// take a position and return always a positive integer between 0 and MAX_TRACK_LENGTH
METHOD PRIVATE TO_POS : DINT
VAR_INPUT
	pos : LREAL;
END_VAR
IF pos < 0 THEN
    TO_POS := LREAL_TO_DINT(pos + CONST.MAX_TRACK_LENGTH);

ELSIF pos >= CONST.MAX_TRACK_LENGTH THEN
    TO_POS := LREAL_TO_DINT(pos) MOD LREAL_TO_DINT(CONST.MAX_TRACK_LENGTH);

ELSE
    TO_POS := LREAL_TO_DINT(pos);

END_IF
END_METHOD

METHOD ToString : STRING
VAR_INPUT
END_VAR
ToString := CONCAT('FB_Mover_', TO_STRING(THIS^._iID));
END_METHOD

END_FUNCTION_BLOCK

// ---- POUs/20_AUTO/Mover/FB_Station.TcPOU
{attribute 'reflection'}
FUNCTION_BLOCK FB_Station IMPLEMENTS IStation, IObject
VAR_INPUT
END_VAR
VAR_OUTPUT
END_VAR
VAR
    _Position          : REFERENCE TO FB_Position;
    _Process           : REFERENCE TO FB_AUT_ABSTRACT;
    _WaitPosOffset     : LREAL; // offset of the station position, should always be negative
    _iMaxWaitingMovers : INT;   // Maximum of waiting mover in front of the station
    _iGroupNumber      : INT;   // The current group member
    _lrOffset          : LREAL; // offset position of this station for a given recipe
    _bSuperTrackNumber : BYTE;  // target number in superTrack

    _ApproachScenario : ApproachScenario_e := ApproachScenario_e.WaitOnFinishedProcess;

    _iID : INT := 0; // instance ID, is set during FB_Init using the value of _iInstanceCounter 
END_VAR
VAR_STAT
    _iInstanceCounter : INT := 1; // instance counter
END_VAR

PROPERTY ApproachScenario : ApproachScenario_e
GET
ApproachScenario := THIS^._ApproachScenario;
END_GET
SET
THIS^._ApproachScenario := ApproachScenario;
END_SET
END_PROPERTY

METHOD Equals : BOOL
VAR_INPUT
    object : ANY;
END_VAR
Equals := THIS = object.pValue;
END_METHOD

METHOD FB_init : BOOL
VAR_INPUT
    bInitRetains      : BOOL; // if TRUE, the retain variables are initialized (warm start / cold start)
    bInCopyCode       : BOOL; // if TRUE, the instance afterwards gets moved into the copy code (online change)
    Position          : REFERENCE TO FB_Position;
    Process           : REFERENCE TO FB_AUT_ABSTRACT;
    WaitPosOffset     : LREAL;
    ApproachScenario  : ApproachScenario_e;
    iMaxWaitingMovers : INT;
	bSuperTrackNumber : BYTE;
END_VAR
THIS^._iID               := THIS^._iInstanceCounter;
THIS^._iInstanceCounter  := THIS^._iInstanceCounter + 1;
THIS^._Position          REF= Position;
THIS^._Process           REF= Process;
THIS^._WaitPosOffset     := WaitPosOffset;
THIS^._ApproachScenario  := ApproachScenario;
THIS^._iMaxWaitingMovers := iMaxWaitingMovers;
THIS^._bSuperTrackNumber := bSuperTrackNumber;
END_METHOD

// the maxuimum number of waiting movers at the front of the station
PROPERTY iMaxWaitingMovers : INT
GET
iMaxWaitingMovers := THIS^._iMaxWaitingMovers;
END_GET
SET
THIS^._iMaxWaitingMovers := iMaxWaitingMovers;
END_SET
END_PROPERTY

PROPERTY PUBLIC Offset : LREAL
GET
Offset := THIS^._lrOffset;
END_GET
SET
THIS^._lrOffset := Offset;
END_SET
END_PROPERTY

PROPERTY Position : REFERENCE TO FB_Position
GET
Position REF=_Position;
END_GET
SET
_Position REF=Position;
END_SET
END_PROPERTY

PROPERTY Process : REFERENCE TO FB_AUT_ABSTRACT
GET
Process REF=_Process;
END_GET
SET
_Process REF= Process;
END_SET
END_PROPERTY

METHOD SetWaitPosOffset : REFERENCE TO FB_Station
VAR_INPUT
	WaitPosOffset : LREAL; // offset position from the given station, must be negative
END_VAR
IF _WaitPosOffset < 0 THEN
    _WaitPosOffset := WaitPos;
END_IF

SetWaitPosOffset REF= THIS^;
END_METHOD

PROPERTY SuperTrackNumber : BYTE
GET
SuperTrackNumber := THIS^._bSuperTrackNumber;
END_GET
END_PROPERTY

METHOD ToString : STRING
VAR_INPUT
END_VAR
VAR_INST
END_VAR
ToString := CONCAT('FB_Station_', TO_STRING(THIS^._iID));
END_METHOD

PROPERTY PUBLIC WaitPos : LREAL
GET
WaitPos := _WaitPosOffset + this^._Position.lrWorkPosition;
END_GET
SET
IF WaitPos < THIS^._Position.lrWorkPosition THEN
    _WaitPosOffset := WaitPos - THIS^._Position.lrWorkPosition;
END_IF
END_SET
END_PROPERTY

END_FUNCTION_BLOCK

// ---- POUs/20_AUTO/Mover/FB_Position.TcPOU
(*
    1D Position class, used to express a given position
	Since the position is in lreal format, you should
	always give a left and a right margin so the isInPosition
	flag will stay stable (beacause we cannot use the = 
	operator on lreal! )
*)
FUNCTION_BLOCK FB_Position IMPLEMENTS IObject
VAR_INPUT
END_VAR
VAR_OUTPUT
END_VAR
VAR
    _lrWorkPosition    : LREAL;      // Work position, use this to give a position
    _lrWorkLeftMargin  : LREAL := 0; // The RELATIVE left position from the work position, need to be POSITIVE
    _lrWorkRightMargin : LREAL := 0; // The RELATIVE right position from the work position, need to be POSITIVE

    _iID : INT := 0; // instance ID, is set during FB_Init using the value of _iInstanceCounter 
END_VAR
VAR_STAT
    _iInstanceCounter : INT := 1; // instance counter
END_VAR

METHOD Equals : BOOL
VAR_INPUT
    object : ANY;
END_VAR
Equals := THIS = object.pValue;
END_METHOD

METHOD FB_init : BOOL
VAR_INPUT
    bInitRetains : BOOL; // if TRUE, the retain variables are initialized (warm start / cold start)
    bInCopyCode  : BOOL; // if TRUE, the instance afterwards gets moved into the copy code (online change)

    lrWorkPosition    : LREAL;      // Work position, use this to give a position
    lrWorkLeftMargin  : LREAL := 0; // The RELATIVE left position from the work position, need to be POSITIVE 
    lrWorkRightMargin : LREAL := 0; // The RELATIVE right position from the work position, need to be POSITIVE
END_VAR
THIS^._iID := THIS^._iInstanceCounter;
THIS^._iInstanceCounter := THIS^._iInstanceCounter +1;
THIS^._lrWorkPosition    := lrWorkPosition;
THIS^._lrWorkLeftMargin  := lrWorkLeftMargin;
THIS^._lrWorkRightMargin := lrWorkRightMargin;
END_METHOD

METHOD isInPos : BOOL
VAR_INPUT
	lrGivenPos : LREAL; // position to test
END_VAR
isInPos := FALSE;

IF ((
    lrGivenPos >= (THIS^._lrWorkPosition - THIS^._lrWorkLeftMargin)) AND
    (lrGivenPos <= (THIS^._lrWorkPosition + THIS^._lrWorkRightMargin)))
    THEN
    isInPos := TRUE;
END_IF
END_METHOD

PROPERTY lrWorkPosition : LREAL
GET
lrWorkPosition := this^._lrWorkPosition;
END_GET
END_PROPERTY

METHOD ToString : STRING
VAR_INPUT
END_VAR
VAR
END_VAR
ToString := CONCAT('FB_Position_', TO_STRING(THIS^._iID));
END_METHOD

END_FUNCTION_BLOCK

// ---- POUs/20_AUTO/ST100/FB_AUT_ABSTRACT.TcPOU
FUNCTION_BLOCK PUBLIC FB_AUT_ABSTRACT IMPLEMENTS IProcessSampleMover
    (****************************************************************************)
    (*	POU_AUT_zxx			Bausteinaufrufe Station	zxx							*)
    (*	Status				ungetestet											*)
    (*  Version:			1.0													*)
    (*	Beschrieb:																*)
    (*																			*)
    (*	Abläufe:			FB_ABLzxxA		Hauptablauf							*)
    (*																			*)
    (*																			*)
    (* 	25.09.2019/Dj															*)
    (****************************************************************************)
    (*	dd.mm.yyyy   KZ    x.y			Beschrieb								*)
    (****************************************************************************)
VAR_INPUT
    (* standart Eingänge *)
    xIN_Init       : BOOL;    // Initialisieren	
    xIN_Quit       : BOOL;    // Fehler quittieren 
    xIN_Start      : BOOL;    // Schrittkette Starten
    xIN_Step       : BOOL;    // Schrittkette Starten/Nachster Schritt
    xIN_ManuCycle  : BOOL;    // Zylus Manuell Starten
    xIN_AlarmAktiv : BOOL;    // Alarm aktiv 
    xIN_DryCycle   : BOOL;    // Fahren ohne Teile 
    enIN_State     : enState; // Status Anlage/Zelle 
    tIN_Timeout    : TIME;    // Timout 
    xIN_On         : BOOL;    // Station eingeschaltet 

    (* spezifische Eingänge *)

END_VAR
VAR_OUTPUT
    (* standart Ausgänge *)
    xOUT_InitDone : BOOL; // fertig initialisiert
    xOUT_Done     : BOOL; // alle Abläufe fertig
    xOUT_Ready    : BOOL; // Station ist bereit (wartet auf Start)
    xOUT_ErrFlag  : BOOL; // Error Flag   
    xOUT_Wait     : BOOL; // alle Abläufe warten
    xOUT_AlarmST  : BOOL; // Station hat Alarm

    (* spezifische Ausgänge *)

END_VAR
VAR

    (* Flags *)
    xReset     : BOOL; // Schrittketten zurücksetzen
    xManuCycle : BOOL; // Manueller Zylus aktiv	
    xNextStep  : BOOL; // Nächster Schritt erlaubt	

    xDummy : BOOL := TRUE; // Platzhalter		

    i : INT;

    _iID : INT := 0; // instance ID, is set during FB_Init using the value of _iInstanceCounter 

    _ProcessExecution : ProcessExecution_e := ProcessExecution_e.ExecuteImmediately;

    _Mover            : REFERENCE TO FB_Mover;
    _xMoverShouldLeave : BOOL; // flag to synchronise process and MoverMan, MoverMan needs to call TakeMover() to reset this flag

END_VAR
VAR_STAT
    _iInstanceCounter : INT := 1; // instance counter
END_VAR

METHOD Equals : BOOL
VAR_INPUT
    object : ANY;
END_VAR
Equals := THIS = object.pValue;
END_METHOD

METHOD FB_init : BOOL
VAR_INPUT
	bInitRetains : BOOL; // if TRUE, the retain variables are initialized (warm start / cold start)
	bInCopyCode : BOOL;  // if TRUE, the instance afterwards gets moved into the copy code (online change)
END_VAR
THIS^._iID := THIS^._iInstanceCounter;
THIS^._iInstanceCounter := THIS^._iInstanceCounter +1;
END_METHOD

METHOD GiveMover : IProcessSampleMover
VAR_INPUT
	mover : REFERENCE TO FB_Mover;
END_VAR
THIS^._Mover REF= mover;
END_METHOD

(* % of completion of the process *)
PROPERTY iCompletionPC : INT
GET
END_GET
END_PROPERTY

(* Process time, expressed in milisecond *)
PROPERTY iProcessTimeMili_1 : DINT
GET
END_GET
SET
END_SET
END_PROPERTY

(* Process time, expressed in milisecond *)
PROPERTY iProcessTimeMili_2 : DINT
GET
END_GET
SET
END_SET
END_PROPERTY

PROPERTY Mover : REFERENCE TO FB_Mover
GET
Mover REF= THIS^._Mover;
END_GET
SET
THIS^._Mover REF= Mover;
END_SET
END_PROPERTY

PROPERTY PUBLIC ProcessExecution : ProcessExecution_e
GET
ProcessExecution := THIS^._ProcessExecution;
END_GET
SET
THIS^._ProcessExecution := ProcessExecution;
END_SET
END_PROPERTY

METHOD TakeMover : IProcessSampleMover
THIS^.Mover REF= 0;
THIS^._xMoverShouldLeave := FALSE;
END_METHOD

METHOD ToString : STRING
VAR_INPUT
END_VAR
VAR
END_VAR
ToString := CONCAT('FB_AUT_ABSTRACT_', TO_STRING(THIS^._iID));
END_METHOD

PROPERTY xBusy : BOOL
GET
END_GET
SET
END_SET
END_PROPERTY

PROPERTY xDone : BOOL
GET
END_GET
END_PROPERTY

PROPERTY xMoverPathFree : BOOL
GET
END_GET
END_PROPERTY

PROPERTY xMoverShouldLeave : BOOL
GET
END_GET
END_PROPERTY

END_FUNCTION_BLOCK

// ---- POUs/20_AUTO/Mover/FB_StationMan.TcPOU
FUNCTION_BLOCK FB_StationMan IMPLEMENTS IObject
VAR_INPUT
END_VAR
VAR_OUTPUT
END_VAR
VAR
    // a null terminated array of working station
    _WorkStationList : ARRAY[1..CONST.STATION_NUMBER] OF POINTER TO FB_Station;
    _SelGroupList    : ARRAY[1..CONST.STATION_NUMBER] OF INT; // hold all station group number of selected station
    _PieceHolder     : REFERENCE TO FB_PieceHolderMover;

    _GroupList : ARRAY[1..CONST.MAX_GROUP] OF FB_Group;

    _iID : INT := 0; // instance ID, is set during FB_Init using the value of _iInstanceCounter 
END_VAR
VAR_STAT
    _iInstanceCounter : INT := 1; // instance counter
END_VAR

// Apply a given station set
// This will build all the needed groups
METHOD PUBLIC ApplyNewPath : BOOL
VAR_INPUT
    // The full station list of the application
    StationList : POINTER TO ARRAY[1..CONST.STATION_NUMBER] OF FB_Station;
    // Used to determine which station is used
    SelStationList : POINTER TO ARRAY[1..CONST.STATION_NUMBER] OF INT;
    PieceHolder    : REFERENCE TO FB_PieceHolderMover;
END_VAR
VAR
    i                 : INT;
    selStationCounter : INT := 1;
END_VAR
FOR i := 1 TO const.STATION_NUMBER BY 1 DO
    IF SelStationList^[i] >= 0 THEN
        THIS^._WorkStationList[selStationCounter] := ADR(StationList^[i]);
        THIS^._SelGroupList[selStationCounter]    := SelStationList^[i];

        selStationCounter := selStationCounter + 1;
    END_IF
END_FOR

FOR selStationCounter := selStationCounter TO CONST.STATION_NUMBER BY 1 DO
    THIS^._WorkStationList[selStationCounter] := 0;
    THIS^._SelGroupList[selStationCounter]    := -1;
END_FOR

THIS^._PieceHolder REF= PieceHolder;
THIS^.SetGroupMembers(StationList, SelStationList);
END_METHOD

METHOD Equals : BOOL
VAR_INPUT
    object : ANY;
END_VAR
Equals := THIS = object.pValue;
END_METHOD

METHOD FB_init : BOOL
VAR_INPUT
    bInitRetains : BOOL; // if TRUE, the retain variables are initialized (warm start / cold start)
    bInCopyCode  : BOOL; // if TRUE, the instance afterwards gets moved into the copy code (online change)

    // The full station list of the application
    StationList : POINTER TO ARRAY[1..CONST.STATION_NUMBER] OF FB_Station;
    // Used to determine which station is used
    SelStationList : POINTER TO ARRAY[1..CONST.STATION_NUMBER] OF INT;
    PieceHolder    : REFERENCE TO FB_PieceHolderMover;
END_VAR
VAR
END_VAR
THIS^._iID              := THIS^._iInstanceCounter;
THIS^._iInstanceCounter := THIS^._iInstanceCounter + 1;

THIS^.ApplyNewPath(StationList, SelStationList, PieceHolder);
END_METHOD

// Return the closest station using the station position 
// First we search if we are in range with our set of station
// then, if no station are in our range, we give the nearest next
// station
METHOD PRIVATE FindCloserStationIndex : INT
VAR_INPUT
    CurrentPosition : LREAL;
END_VAR
VAR
    i : INT;
END_VAR
FindCloserStationIndex := -1;

// First we check if we are not in range of a station from our set
FOR i := 1 TO CONST.STATION_NUMBER BY 1 DO
    IF 0 <> THIS^._WorkStationList[i] THEN
        IF THIS^._WorkStationList[i]^.Position.isInPos(CurrentPosition) THEN
            FindCloserStationIndex := i;
            RETURN;
        END_IF
    END_IF
END_FOR

// Then, if no station are in the range, we give the most nearest station, if possible
FOR i := 1 TO CONST.STATION_NUMBER BY 1 DO
    IF 0 <> THIS^._WorkStationList[i] THEN
        IF __ISVALIDREF(THIS^._WorkStationList[i]^.Position) AND
           THIS^._WorkStationList[i]^.Position.lrWorkPosition > CurrentPosition THEN
            FindCloserStationIndex := i;
            EXIT;
        END_IF
    END_IF
END_FOR
END_METHOD

// Return the next station to visit
METHOD GetNextStation : REFERENCE TO FB_Station
VAR_INPUT
    CurrentStation : REFERENCE TO FB_Station;
END_VAR
VAR
    CurrStationIndex : INT;
	NextStationIndex : INT;
END_VAR
GetNextStation   REF= CurrentStation;
CurrStationIndex := THIS^.GetStationIndex(CurrentStation);
NextStationIndex := CurrStationIndex;

IF CurrStationIndex > 0 THEN

    IF THIS^._SelGroupList[CurrStationIndex] > 0 THEN
        // We search for a station which is not from the same group
        WHILE THIS^._SelGroupList[CurrStationIndex] = THIS^._SelGroupList[NextStationIndex] DO
			// We have to use NextStationIndex otherwise we stay with the 2 same
			// station over and over again
            NextStationIndex := THIS^.GetNextStationIndex(NextStationIndex);
            GetNextStation   REF= THIS^._WorkStationList[NextStationIndex]^;
        END_WHILE
    ELSE
        NextStationIndex := THIS^.GetNextStationIndex(CurrStationIndex);
        GetNextStation   REF= THIS^._WorkStationList[NextStationIndex]^;
    END_IF

    // We take a look of the group member and then set the corresponding station
    IF THIS^._SelGroupList[NextStationIndex] > 0 THEN
        GetNextStation REF= THIS^._GroupList[THIS^._SelGroupList[NextStationIndex]].GetNextStation();
    END_IF

    // when the current is not on the list, we try to move to the nearest
    // but only on the positive direction
ELSE
    CurrStationIndex := THIS^.FindCloserStationIndex(CurrentStation.Position.lrWorkPosition);

    IF CurrStationIndex > 0 THEN
        GetNextStation REF= THIS^._WorkStationList[CurrStationIndex]^;

    ELSE
        GetNextStation REF= THIS^._WorkStationList[1]^;

    END_IF
END_IF
END_METHOD

// Return the next station index in the ring buffer of station
METHOD PRIVATE GetNextStationIndex : INT
VAR_INPUT
	CurrStationIndex : INT;
END_VAR
IF CurrStationIndex >= CONST.STATION_NUMBER THEN
    GetNextStationIndex := 1;

ELSIF THIS^._WorkStationList[CurrStationIndex + 1] = 0 THEN
    GetNextStationIndex := 1;

ELSE
    GetNextStationIndex := CurrStationIndex + 1;
END_IF
END_METHOD

// Get the next station with a valid process. If nothing is found, we 
// simply return to the first station (this should be never the case
// since your machine will be useless...)
METHOD GetNextStationWithProcess : REFERENCE TO FB_Station
VAR_INPUT
    CurrentStation : REFERENCE TO FB_Station;
END_VAR
VAR
    // search station with process algorithme
    iSearchNext        : INT; // incremtal variable used to search in a set of next station
    iTempSearchStation : INT; // incremtal variable used to search in a set of next station
    tempStation        : REFERENCE TO FB_Station;
END_VAR
// If nothing found, we return to the first station
GetNextStationWithProcess REF= THIS^._WorkStationList[1]^;

IF __ISVALIDREF(CurrentStation) THEN
    iSearchNext := 1;

    WHILE iSearchNext < CONST.STATION_NUMBER DO
        tempStation REF= THIS^.GetNextStation(CurrentStation);

        IF __ISVALIDREF(tempStation) AND_THEN __ISVALIDREF(tempStation.Process) THEN
            GetNextStationWithProcess REF= tempStation;
            EXIT;
        END_IF

        iSearchNext := iSearchNext + 1;

    END_WHILE
END_IF
END_METHOD

METHOD GetStartStation : POINTER TO FB_Station
VAR_INPUT
    CurrentPosition : LREAL;
END_VAR
VAR
    CurrStationIndex : INT;
END_VAR
//GetStartStation := THIS^._WorkStationList[1];
CurrStationIndex := THIS^.FindCloserStationIndex(CurrentPosition);

IF CurrStationIndex > 0 THEN
    GetStartStation := THIS^._WorkStationList[CurrStationIndex];

ELSE
    GetStartStation := THIS^._WorkStationList[1];

END_IF
END_METHOD

// return the index of a given station, If the index is -1, no station where found
METHOD PRIVATE GetStationIndex : INT
VAR_INPUT
    Station : REFERENCE TO FB_Station;
END_VAR
VAR
    i : INT;
END_VAR
GetStationIndex := -1;

FOR i := 1 TO CONST.STATION_NUMBER BY 1 DO
    IF Station.Equals(THIS^._WorkStationList[i]^) THEN
        GetStationIndex := i;
        EXIT;
    END_IF
END_FOR
END_METHOD

METHOD IsProcessUsed : BOOL
VAR_INPUT
	process : REFERENCE TO FB_AUT_ABSTRACT;
END_VAR
VAR
	i : INT;
END_VAR
FOR i := 1 TO CONST.STATION_NUMBER BY 1 DO
	IF (0 <> THIS^._WorkStationList[i]) AND_THEN __ISVALIDREF(THIS^._WorkStationList[i]^.Process) THEN
		IF THIS^._WorkStationList[i]^.Process.Equals(process) THEN
			IsProcessUsed := TRUE;
			EXIT; 
		END_IF
	END_IF
END_FOR
END_METHOD

PROPERTY PieceHolder : REFERENCE TO FB_PieceHolderMover
GET
PieceHolder REF= _PieceHolder;
END_GET
SET
_PieceHolder REF= PieceHolder;
END_SET
END_PROPERTY

METHOD SetGroupMembers : REFERENCE TO FB_Group
VAR_INPUT
    // The full station list of the application
    StationList : POINTER TO ARRAY[1..CONST.STATION_NUMBER] OF FB_Station;
    SelStationList : POINTER TO ARRAY[1..CONST.STATION_NUMBER] OF INT;
END_VAR
VAR
    i : INT;
END_VAR
FOR i := 1 TO CONST.STATION_NUMBER BY 1 DO
    IF SelStationList^[i] > 0 AND SelStationList^[i] <= CONST.MAX_GROUP THEN
        THIS^._GroupList[SelStationList^[i]].AddStation(StationList^[i]);
    END_IF
END_FOR
END_METHOD

METHOD ToString : STRING
VAR_INPUT
END_VAR
VAR
END_VAR
ToString := CONCAT('FB_StationMan_', TO_STRING(THIS^._iID));
END_METHOD

END_FUNCTION_BLOCK

// ---- POUs/20_AUTO/Mover/FB_Group.TcPOU
// Create station group and manage shuttle behaviour 
FUNCTION_BLOCK FB_Group IMPLEMENTS IObject
VAR_INPUT
END_VAR
VAR_OUTPUT
END_VAR
VAR
    _GroupNumber : INT; // group number

    _StationList : ARRAY[1..CONST.MAX_STATION_PER_GROUP] OF POINTER TO FB_Station; // Array of member station member

    _LastVisitedIndex : INT; // Last visited station index
    _MaxStationList   : INT; // The current maximum of station in this group. 0 means no station are present
	
	_iID : INT := 0; // instance ID, is set during FB_Init using the value of _iInstanceCounter 
END_VAR
VAR_STAT
	_iInstanceCounter : INT; // instance counter
END_VAR

METHOD AddStation : REFERENCE TO FB_Group
VAR_INPUT
    station : REFERENCE TO FB_Station;
END_VAR
IF THIS^._MaxStationList < CONST.MAX_STATION_PER_GROUP THEN
    THIS^._MaxStationList                     := THIS^._MaxStationList + 1;
    THIS^._StationList[THIS^._MaxStationList] := ADR(station);
ELSE
    ASSERT(0);
END_IF
END_METHOD

METHOD Equals : BOOL
VAR_INPUT
    object : ANY;
END_VAR
Equals := THIS = object.pValue;
END_METHOD

METHOD FB_init : BOOL
VAR_INPUT
    bInitRetains : BOOL; // if TRUE, the retain variables are initialized (warm start / cold start)
    bInCopyCode  : BOOL; // if TRUE, the instance afterwards gets moved into the copy code (online change)
END_VAR
THIS^._iInstanceCounter := THIS^._iInstanceCounter + 1;
THIS^._iID              := THIS^._iInstanceCounter;

THIS^._MaxStationList   := 0;
THIS^._LastVisitedIndex := 1; // the last station is set to the first

IF THIS^._iID <= CONST.MAX_GROUP THEN
    THIS^._GroupNumber := THIS^._iID;
ELSE
    ASSERT(0);
END_IF
END_METHOD

// The next station is always the one before the last visited
METHOD GetNextStation : REFERENCE TO FB_Station
VAR_INPUT
END_VAR
(* Note about this algorithme :
 * The goal of this algorithm is to divide equaly the use of each station
 * so the wear of station is the same. Other algorithm can be implemented 
 * if needed.
*)
IF THIS^._LastVisitedIndex <= 1 THEN
    THIS^._LastVisitedIndex := THIS^._MaxStationList;
ELSE
    THIS^._LastVisitedIndex := THIS^._LastVisitedIndex - 1;
END_IF

IF THIS^._LastVisitedIndex <= 0 THEN
	ASSERT(0); // should never be 0 since index goes from 1 to max station index
	THIS^._LastVisitedIndex := 1;
END_IF

GetNextStation REF= THIS^._StationList[THIS^._LastVisitedIndex]^;
END_METHOD

PROPERTY GroupNumber : INT
GET
GroupNumber := this^._GroupNumber;
END_GET
END_PROPERTY

METHOD ToString : STRING
VAR_INPUT
END_VAR
ToString := CONCAT('FB_Station_', TO_STRING(THIS^._iID));
END_METHOD

END_FUNCTION_BLOCK

// ---- POUs/10_HMI/_14_STATE.TcPOU
PROGRAM _14_STATE
(****************************************************************************)
//STATE PROGRAMM
//	- Control Buttons
//	- Status Anlage
//
//	05.09.2019/Dj
//
//	Version:
(****************************************************************************)
VAR
    fb_State        :   FB_State;       //Status der Maschine
	sStateDbg		: STRING;		// enState but in string format
		
	//Control Buttons
	_FB_btAUTO	: FB_BUTTON;
	_FB_btSTEP	: FB_BUTTON;
	_FB_btEND	: FB_BUTTON;
	_FB_btMANU	: FB_BUTTON;
	_FB_btINIT	: FB_BUTTON;
	_FB_btSTOP	: FB_BUTTON;
	_FB_btLEER	: FB_BUTTON;
	_FB_btQUIT	: FB_BUTTON;
	_FB_btSTART	: FB_BUTTON;
END_VAR

//****************************************************************************
// 	CONTROL BUTTONS
//****************************************************************************
//	AUTO 
_FB_btAUTO(pbtIN  := ADR(HMI.btArMain[0]),
           xINdis := (HMI.enState < enState.StateREADY),
           xINon  := (HMI.enState = enState.StateAUTO),
           xINerr := FALSE);

//STEP
_FB_btSTEP(pbtIN  := ADR(HMI.btArMain[1]),
           xINdis := (HMI.enState < enState.StateREADY),
           xINon  := (HMI.enState = enState.StateSTEP),
           xINerr := FALSE);

//END
_FB_btEND(pbtIN  := ADR(HMI.btArMain[2]),
          xINdis := (HMI.enState < enState.StateREADY),
          xINon  := (HMI.enState = enState.StateEND),
          xINerr := FALSE);

//MANU
_FB_btMANU(pbtIN  := ADR(HMI.btArMain[3]),
           xINdis := (HMI.enState > enState.StateSTEP) OR
                     (HMI.enState = enState.StateALARM) OR
                     (HMI.enState < enState.StateAIRon),
           xINon  := (HMI.enState = enState.StateMANU),
           xINerr := FALSE);

//INIT
_FB_btINIT(pbtIN  := ADR(HMI.btArMain[4]),
           xINdis := (HMI.enState < enState.StateENGIZED),
           xINon  := (HMI.enState = enState.StateINIT),
           xINerr := FALSE);

//STOP
_FB_btSTOP(pbtIN  := ADR(HMI.btArMain[5]),
           xINdis := (HMI.enState < enState.StateENGIZED),
           xINon  := FALSE,
           xINerr := FALSE);

//LEERFAHREN
_FB_btLEER(pbtIN  := ADR(HMI.btArMain[6]),
           xINdis := FALSE,
           xINon  := FALSE,
           xINerr := FALSE);

//QUIT
_FB_btQUIT(pbtIN  := ADR(HMI.btArMain[7]),
           xINdis := FALSE,
           xINon  := FALSE,
           xINerr := HMI.xAlarm);

//START
_FB_btSTART(pbtIN  := ADR(HMI.btArMain[9]),
            xINdis := HMI.enState < enState.StateREADY,
            xINon  := HMI.btArMain[9].on,
            xINerr := FALSE);

//****************************************************************************
// 	STATE FB
//****************************************************************************
fb_State(xIN_AutoInit   := TRUE,
         xIN_DoRef      := FALSE,
         xIN_ENERGIE    := TRUE,
         xIN_AIR        := HMI.xAIRon,
         xIN_EINRICHTEN :=,
         xIN_AUTO       := HMI.btArMain[0].rtrig,
         xIN_STEP       := HMI.btArMain[1].rtrig,
         xIN_CYCLE      := HMI.btArMain[2].rtrig,
         xIN_MANU       := HMI.btArMain[3].rtrig,
         xIN_INIT       := HMI.btArMain[4].rtrig,
         xIN_STOP       := HMI.btArMain[5].rtrig,
         xIN_LEER       := HMI.btArMain[6].rtrig,
         xIN_InitEND    := PRG.st105_aut.xOUT_InitDone AND
                           PRG.st110_aut.xOUT_InitDone AND
                           PRG.st115_aut.xOUT_InitDone AND
                           PRG.st120_aut.xOUT_InitDone AND
                           PRG.st125_aut.xOUT_InitDone AND
                           PRG.st130_aut.xOUT_InitDone AND
                           PRG.st135_aut.xOUT_InitDone AND
                           PRG.st140_aut.xOUT_InitDone AND
                           PRG.st145_aut.xOUT_InitDone AND
                           PRG.st150_aut.xOUT_InitDone AND
                           PRG.st155_aut.xOUT_InitDone AND
                           PRG.st160_aut.xOUT_InitDone AND
                           PRG.st165_aut.xOUT_InitDone AND
                           PRG.st170_aut.xOUT_InitDone AND
                           PRG.st175_aut.xOUT_InitDone AND
                           PRG.st176_aut.xOUT_InitDone AND
                           PRG.st180_aut.xOUT_InitDone AND
                           PRG.st185_aut.xOUT_InitDone,
         xIN_ALARM := PRG.st105_aut.xOUT_ErrFlag AND
                      PRG.st110_aut.xOUT_errFlag AND
                      PRG.st115_aut.xOUT_errFlag AND
                      PRG.st120_aut.xOUT_errFlag AND
                      PRG.st125_aut.xOUT_errFlag AND
                      PRG.st130_aut.xOUT_errFlag AND
                      PRG.st135_aut.xOUT_errFlag AND
                      PRG.st140_aut.xOUT_errFlag AND
                      PRG.st145_aut.xOUT_errFlag AND
                      PRG.st150_aut.xOUT_errFlag AND
                      PRG.st155_aut.xOUT_errFlag AND
                      PRG.st160_aut.xOUT_errFlag AND
                      PRG.st165_aut.xOUT_errFlag AND
                      PRG.st170_aut.xOUT_errFlag AND
                      PRG.st175_aut.xOUT_errFlag AND
                      PRG.st176_aut.xOUT_errFlag AND
                      PRG.st180_aut.xOUT_errFlag AND
                      PRG.st185_aut.xOUT_errFlag AND
                      (PRG.st105_aut.xOUT_ErrFlag OR PRG.st105_aut.xOUT_wait) AND
                      (PRG.st110_aut.xOUT_errFlag OR PRG.st110_aut.xOUT_wait) AND
                      (PRG.st115_aut.xOUT_errFlag OR PRG.st115_aut.xOUT_wait) AND
                      (PRG.st120_aut.xOUT_errFlag OR PRG.st120_aut.xOUT_wait) AND
                      (PRG.st125_aut.xOUT_errFlag OR PRG.st125_aut.xOUT_wait) AND
                      (PRG.st130_aut.xOUT_errFlag OR PRG.st130_aut.xOUT_wait) AND
                      (PRG.st135_aut.xOUT_errFlag OR PRG.st135_aut.xOUT_wait) AND
                      (PRG.st140_aut.xOUT_errFlag OR PRG.st140_aut.xOUT_wait) AND
                      (PRG.st145_aut.xOUT_errFlag OR PRG.st145_aut.xOUT_wait) AND
                      (PRG.st150_aut.xOUT_errFlag OR PRG.st150_aut.xOUT_wait) AND
                      (PRG.st155_aut.xOUT_errFlag OR PRG.st155_aut.xOUT_wait) AND
                      (PRG.st160_aut.xOUT_errFlag OR PRG.st160_aut.xOUT_wait) AND
                      (PRG.st165_aut.xOUT_errFlag OR PRG.st165_aut.xOUT_wait) AND
                      (PRG.st170_aut.xOUT_errFlag OR PRG.st170_aut.xOUT_wait) AND
                      (PRG.st175_aut.xOUT_errFlag OR PRG.st175_aut.xOUT_wait) AND
                      (PRG.st176_aut.xOUT_errFlag OR PRG.st176_aut.xOUT_wait) AND
                      (PRG.st180_aut.xOUT_errFlag OR PRG.st180_aut.xOUT_wait) AND
                      (PRG.st185_aut.xOUT_errFlag OR PRG.st185_aut.xOUT_wait),
         xIN_LastDone := (PRG.st105_aut.xOUT_Done OR PRG.st105_aut.xout_InitDone) AND
                         (PRG.st110_aut.xOUT_Done OR PRG.st110_aut.xout_InitDone) AND
                         (PRG.st115_aut.xOUT_Done OR PRG.st115_aut.xout_InitDone) AND
                         (PRG.st120_aut.xOUT_Done OR PRG.st120_aut.xout_InitDone) AND
                         (PRG.st125_aut.xOUT_Done OR PRG.st125_aut.xout_InitDone) AND
                         (PRG.st130_aut.xOUT_Done OR PRG.st130_aut.xout_InitDone) AND
                         (PRG.st135_aut.xOUT_Done OR PRG.st135_aut.xout_InitDone) AND
                         (PRG.st140_aut.xOUT_Done OR PRG.st140_aut.xout_InitDone) AND
                         (PRG.st145_aut.xOUT_Done OR PRG.st145_aut.xout_InitDone) AND
                         (PRG.st150_aut.xOUT_Done OR PRG.st150_aut.xout_InitDone) AND
                         (PRG.st155_aut.xOUT_Done OR PRG.st155_aut.xout_InitDone) AND
                         (PRG.st160_aut.xOUT_Done OR PRG.st160_aut.xout_InitDone) AND
                         (PRG.st165_aut.xOUT_Done OR PRG.st165_aut.xout_InitDone) AND
                         (PRG.st170_aut.xOUT_Done OR PRG.st170_aut.xout_InitDone) AND
                         (PRG.st175_aut.xOUT_Done OR PRG.st175_aut.xout_InitDone) AND
                         (PRG.st176_aut.xOUT_Done OR PRG.st176_aut.xout_InitDone) AND
                         (PRG.st180_aut.xOUT_Done OR PRG.st180_aut.xout_InitDone) AND
                         (PRG.st185_aut.xOUT_Done OR PRG.st185_aut.xout_InitDone),
         xIN_WaitFBs := PRG.st105_aut.xOUT_Wait OR
                        PRG.st110_aut.xOUT_Wait OR
                        PRG.st115_aut.xOUT_Wait OR
                        PRG.st120_aut.xOUT_Wait OR
                        PRG.st125_aut.xOUT_Wait OR
                        PRG.st130_aut.xOUT_Wait OR
                        PRG.st135_aut.xOUT_Wait OR
                        PRG.st140_aut.xOUT_Wait OR
                        PRG.st145_aut.xOUT_Wait OR
                        PRG.st150_aut.xOUT_Wait OR
                        PRG.st155_aut.xOUT_Wait OR
                        PRG.st160_aut.xOUT_Wait OR
                        PRG.st165_aut.xOUT_Wait OR
                        PRG.st170_aut.xOUT_Wait OR
                        PRG.st175_aut.xOUT_Wait OR
                        PRG.st176_aut.xOUT_Wait OR
                        PRG.st180_aut.xOUT_Wait OR
                        PRG.st185_aut.xOUT_Wait,
         enINOUT_State => HMI.enState);

sStateDbg := TO_STRING(HMI.enState);

END_PROGRAM

// ---- POUs/20_AUTO/TOOL/SortBubbleLREAL.TcPOU
FUNCTION SortBubbleLREAL : BOOL
VAR_INPUT
    pArray      : POINTER TO LREAL; // Pointer to the array of LREAL
    iStartIndex : INT;
    iStopIndex  : INT;
END_VAR
VAR
    i    : INT;
    j    : INT;
    temp : LREAL;
END_VAR

FOR i := iStartIndex TO iStopIndex BY 1 DO
    FOR j := iStartIndex TO iStopIndex - i -1 BY 1 DO
        IF pArray[j] > pArray[j + 1] THEN
            temp          := pArray[j];
            pArray[j]     := pArray[j + 1];
            pArray[j + 1] := temp;
        END_IF
    END_FOR
END_FOR

END_FUNCTION

// ---- POUs/00_MAIN/_05_FLAGS.TcPOU
PROGRAM _05_FLAGS
(****************************************************************************)
//FLAGS PROGRAMM
//	- Diverse Allgemeine Signale
//
//	04.09.2019/Dj
//
//	Version:
(****************************************************************************)
VAR_INPUT
	xIN_AIR			: 	BOOL;				//Luftdruck
	xIN_btRES_TEMP	:	structButton;		//BUTTON ResetCounter
END_VAR
VAR
	TOF_AirOFF		: 	TOF;				//Air NIO
	TON_btReset		:	TON;				//Reset Taste gedrückt
	
    _FB_Lampe		:   FB_LampeBNI007F;	//Lampe Balluf BN007F
	
	_FB_btRESET		: 	FB_BUTTON;			//Reset Temp Counter
	
END_VAR

//--------------------------------------------------------------------------
//Air ON
//--------------------------------------------------------------------------
TOF_AirOFF(IN:=xIN_AIR , PT:=T#500MS);
HMI.xAIRon	:= TOF_AirOFF.Q;

//--------------------------------------------------------------------------
//Reset Counter	
//--------------------------------------------------------------------------
//Button
_FB_btRESET(pbtIN:= ADR(xIN_btRES_TEMP),
	xINdis:= FALSE, 
	xINon:= (PERS.udiTempNOK=0) AND (PERS.udiTempOK=0), 
	xINerr:= FALSE);
TON_btReset(IN:=xIN_btRES_TEMP.press, PT:=T#1.5S);
//Reset
IF TON_btReset.Q THEN
	PERS.udiTempNOK:=0;
	PERS.udiTempOK:=0;
END_IF

//--------------------------------------------------------------------------
//Flanken
//--------------------------------------------------------------------------

END_PROGRAM

// ---- POUs/10_HMI/_10_HMI.TcPOU
PROGRAM _10_HMI
(****************************************************************************)
//HMI PROGRAMM
//	- HMI RELEVANTE Signale und Funktionen
//
//	04.09.2019/Dj
//
//	Version:
(****************************************************************************)

VAR
	//Startup HMI-Panel
	TON_startup		:	TON;
	
	//Reset Counter
	TON_ResetCounter			: 	TON;			// Reset Temparary Counter
	
	//Ticker
	TICK6M						:	TP;				// Ticker for Operating Hours
	TICK6M_						: 	TP;
	x_TICK6M					:	BOOL;	
	BLINK_500					: 	TP;				// Ticker for Operating Hours
	BLINK_500_					: 	TP;
	x_BLINK_500					: 	BOOL;
	
	BLINK_100					: 	TP;				// Ticker for Operating Hours
	BLINK_100_					: 	TP;
	x_BLINK_100					: 	BOOL;	
	
	//Cycle Time
	_FB_SystemTime				: 	GETSYSTEMTIME;
	dw_ActTime					: 	DWORD;
	
	//Lampen
	_FB_LAMPE					: FB_LampeBNI007F;
	
	
	//Alarmlog
	iCount6h					: 	INT;			//6h Ticker (für AlarmLOG)
	rtNOTAUS					:	R_TRIG;			//Trigger 6h	
	
	//Divers
	idx							:	INT;			//Index
END_VAR

//***********************************************************************************************)
//Startup Terminal
//***********************************************************************************************)
TON_Startup(IN := TRUE, PT := T#5S);

//***********************************************************************************************)
//Parameter ÜBERPRÜFEN
//***********************************************************************************************)
_11_PAR_CHK();

//***********************************************************************************************)
//State
//***********************************************************************************************)
_14_STATE();

//***********************************************************************************************)
//Lampen
//***********************************************************************************************)
_FB_LAMPE(enIN_State     := HMI.enState,
          xIN_AlarmAktiv := PRG.st105_aut.xOUT_ErrFlag OR
                            PRG.st110_aut.xOUT_errFlag OR
                            PRG.st115_aut.xOUT_errFlag OR
                            PRG.st120_aut.xOUT_errFlag OR
                            PRG.st125_aut.xOUT_errFlag OR
                            PRG.st130_aut.xOUT_errFlag OR
                            PRG.st135_aut.xOUT_errFlag OR
                            PRG.st140_aut.xOUT_errFlag OR
                            PRG.st145_aut.xOUT_errFlag OR
                            PRG.st150_aut.xOUT_errFlag OR
                            PRG.st155_aut.xOUT_errFlag OR
                            PRG.st160_aut.xOUT_errFlag OR
                            PRG.st165_aut.xOUT_errFlag OR
                            PRG.st170_aut.xOUT_errFlag OR
                            PRG.st175_aut.xOUT_errFlag OR
                            PRG.st176_aut.xOUT_errFlag OR
                            PRG.st180_aut.xOUT_errFlag OR
                            PRG.st185_aut.xOUT_errFlag,
          xIN_SafetyError := FALSE,
          xIN_NotAus      := FALSE,
          xIN_Mel1        :=,
          xIN_Mel2        :=,
          xIN_Mel3        :=,
          xIN_Mel4        :=,
          xIN_Mel5        :=,
          xIN_Mel6        :=,
          xIN_Mel7        :=,
          tIN_Meldungen   := T#1000MS,
          tIN_Impuls      := T#500ms,
          xOUT_ErrFlag    =>);

//BALLUFF LAMPE
//OUT.QW194A3:=_FB_LAMPE.wOUT_Lampe;
//OUT.QW194A6:=_FB_LAMPE.wOUT_Lampe;
//OUT.Q194A3_SycStart:=_FB_LAMPE.xOUT_SyncStart;
//OUT.Q194A6_SycStart:=_FB_LAMPE.xOUT_SyncStart;
//OUT.Q194A3_SycImp:=_FB_LAMPE.xOUT_SyncImp;
//OUT.Q194A6_SycImp:=_FB_LAMPE.xOUT_SyncImp;
//LAMPE ENERGIE EIN 
(*
OUT.Q000_LAMP_NRJ:= _10_HMI.x_BLINK_500 AND 
						//Notaus Schalter
						_02_Safety.bArIN_Input[1].4 AND
						_02_Safety.bArIN_Input[2].0 AND	
						_02_Safety.bArIN_Input[2].2 AND
						_02_Safety.bArIN_Input[2].4 AND
						_02_Safety.bArIN_Input[2].6 
					OR (HMI.enState>enState.StateOFF);
					*)

(***********************************************************************************************)
(* HMI Alarme*)
(***********************************************************************************************)
FOR idx := 1 TO 100 BY 1 DO
    HMI.xArAlarmHMI[idx] := HMI.strArALARM[idx].xAlarmOUT;
END_FOR

FOR idx := 1 TO 100 BY 1 DO
    HMI.xArAlarmHMI[idx + 5000] := HMI.strArMSG[idx].xAlarmOUT;
END_FOR

(***********************************************************************************************)
(* Cycle Time *)
(***********************************************************************************************)
_FB_SystemTime(timeLoDW => dw_ActTime, timeHiDW =>);
dw_ActTime := dw_ActTime AND 16#FFFF0000;

(***********************************************************************************************)
(* Operating hours  *)
(***********************************************************************************************)
(* 0.5' Blinker *)
BLINK_500(IN := NOT BLINK_500_.Q, PT := T#500MS, Q => x_BLINK_500);
BLINK_500_(IN := NOT BLINK_500.Q, PT := T#500MS);
(* 0.1' Blinker *)
BLINK_100(IN := NOT BLINK_100_.Q, PT := T#100MS, Q => x_BLINK_100);
BLINK_100_(IN := NOT BLINK_100.Q, PT := T#100MS);
(* 6' Ticker *)
TICK6M(IN := NOT TICK6M_.Q, PT := T#1MS, Q => x_TICK6M);
TICK6M_(IN := NOT TICK6M.Q, PT := t#6m);

(* Operating hours *)
IF TICK6M.Q THEN
    (* AUTO *)
    IF (HMI.enState = enState.StateAUTO) THEN
        PERS.udiCount6Mauto := PERS.udiCount6Mauto + 1;
        IF (PERS.udiCount6Mauto >= 10) THEN
            PERS.udiCount6Mauto := 0;
            PERS.udiCountHauto  := PERS.udiCountHauto + 1;
            IF (PERS.udiCountHauto < 0) THEN
                PERS.udiCountHauto := 0;
            END_IF;
        END_IF;
    END_IF;

    (* TOTAL *)
    PERS.udiCount6Mon := PERS.udiCount6Mon + 1;
    IF (PERS.udiCount6Mon >= 10) THEN
        PERS.udiCount6Mon := 0;
        PERS.udiCountHon  := PERS.udiCountHon + 1;
        IF (PERS.udiCountHon < 0) THEN
            PERS.udiCountHon := 0;
        END_IF;
    END_IF;

    //6h
    iCount6h := iCount6h + 1;
END_IF;

//Alarmlog schreiben nach 6h oder bei NOT-AUS
//rtNOTAUS(CLK:=_02_SAFETY.xOUT_ESout);
IF (iCount6h >= 60) OR rtNOTAUS.Q THEN
    iCount6h        := 0;
    HMI.xWriteALlog := NOT HMI.xWriteALlog;
END_IF;

END_PROGRAM

// ---- POUs/10_HMI/_11_PAR_CHK.TcPOU
PROGRAM _11_PAR_CHK
(****************************************************************************)
//HMI PARAMETER VALIDIEREN
//	- Achsenpositionen gültig
//	- Achse in Position 
//	- Achse Freilauf
//
//	13.09.2019/Dj
//
//	Version:	1.0
(****************************************************************************)
VAR_INPUT
	//Axis01X1
	rIN_TolP_01X1		: REAL;	//Toleranz+ inPOS
	rIN_TolN_01X1		: REAL;	//Toleranz- inPOS
	//Axis01Y2
	rIN_TolP_01Y2		: REAL;	//Toleranz+ inPOS
	rIN_TolN_01Y2		: REAL;	//Toleranz- inPOS
	//Axis01Z3
	rIN_TolP_01Z3		: REAL;	//Toleranz+ inPOS
	rIN_TolN_01Z3		: REAL;	//Toleranz- inPOS
	//Axis02W1
	rIN_TolP_02W1		: REAL;	//Toleranz+ inPOS
	rIN_TolN_02W1		: REAL;	//Toleranz- inPOS
END_VAR
VAR
	bIdx				: BYTE;	//Index
END_VAR
VAR_OUTPUT
	xOUT_Axis01X1valid	: BOOL;	//Axis valid
	xOUT_Axis01Y2valid	: BOOL;	//Axis valid
	xOUT_Axis01Z3valid	: BOOL;	//Axis valid
	xOUT_Axis02W1valid	: BOOL;	//Axis valid
END_VAR

END_PROGRAM

// ---- POUs/20_AUTO/_20_AUTO.TcPOU
PROGRAM
    _20_AUTO
VAR_INPUT
    xIN_Quit   : BOOL;    //Quittieren
    enIN_State : enState; //Status der Maschine 
END_VAR
VAR
    i : INT;

    pFB_Load   : POINTER TO FB_AUT_LOAD;
    pFB_Unload : POINTER TO FB_AUT_UNLOAD;
    pFB_Modify : POINTER TO FB_AUT_MODIFY;
    fbLofad    : FB_AUT_LOAD;
    fb_Unload  : FB_AUT_UNLOAD;
    fb_Modify  : FB_AUT_MODIFY;
    bResult    : BOOL;
END_VAR

//Alarm Allgemein
//POU_ERR_000(xIN_QUIT:=xIN_Quit , pstrArIN_ALARM:=ADR(HMI.strArALARM[1]));
//POU_MSG_000(xIN_QUIT:=xIN_Quit , pstrArIN_ALARM:=ADR(HMI.strArMSG[1]));

//Station01

SIMU.iCompletionHMI[1]           := PRG.st105_aut.iCompletionPC;
PRG.st105_aut.iProcessTimeMili_1 := PERS.iStationTimeDef1[1];
PRG.st105_aut.iProcessTimeMili_2 := PERS.iStationTimeDef2[1];
PRG.st105_aut(xIN_Init       := HMI.enState = enState.StateINIT,
              xIN_Start      := HMI.btArMain[9].press,
              xIN_Step       := HMI.btArMain[1].rtrig,
              xIN_ManuCycle  := FALSE,
              xIN_ManuCycle  := FALSE,
              xIN_Quit       := xIN_Quit,
              xIN_AlarmAktiv := HMI.xAlarm,
              xIN_DryCycle   := FALSE,
              enIN_State     := enIN_State,
              tIN_Timeout    := T#10S,
              xIN_On         := TRUE);

SIMU.iCompletionHMI[2]           := PRG.st110_aut.iCompletionPC;
PRG.st110_aut.iProcessTimeMili_1 := PERS.iStationTimeDef1[2];
PRG.st110_aut.iProcessTimeMili_2 := PERS.iStationTimeDef2[2];
PRG.st110_aut(xIN_Init       := HMI.enState = enState.StateINIT,
              xIN_Start      := HMI.btArMain[9].press,
              xIN_Step       := HMI.btArMain[1].rtrig,
              xIN_ManuCycle  := FALSE,
              xIN_ManuCycle  := FALSE,
              xIN_Quit       := xIN_Quit,
              xIN_AlarmAktiv := HMI.xAlarm,
              xIN_DryCycle   := FALSE,
              enIN_State     := enIN_State,
              tIN_Timeout    := T#10S,
              xIN_On         := TRUE);

SIMU.iCompletionHMI[3]           := PRG.st115_aut.iCompletionPC;
PRG.st115_aut.iProcessTimeMili_1 := PERS.iStationTimeDef1[3];
PRG.st115_aut.iProcessTimeMili_2 := PERS.iStationTimeDef2[3];
PRG.st115_aut(xIN_Init       := HMI.enState = enState.StateINIT,
              xIN_Start      := HMI.btArMain[9].press,
              xIN_Step       := HMI.btArMain[1].rtrig,
              xIN_ManuCycle  := FALSE,
              xIN_ManuCycle  := FALSE,
              xIN_Quit       := xIN_Quit,
              xIN_AlarmAktiv := HMI.xAlarm,
              xIN_DryCycle   := FALSE,
              enIN_State     := enIN_State,
              tIN_Timeout    := T#10S,
              xIN_On         := TRUE);

SIMU.iCompletionHMI[4]           := PRG.st120_aut.iCompletionPC;
PRG.st120_aut.iProcessTimeMili_1 := PERS.iStationTimeDef1[4];
PRG.st120_aut.iProcessTimeMili_2 := PERS.iStationTimeDef2[4];
PRG.st120_aut(xIN_Init       := HMI.enState = enState.StateINIT,
              xIN_Start      := HMI.btArMain[9].press,
              xIN_Step       := HMI.btArMain[1].rtrig,
              xIN_ManuCycle  := FALSE,
              xIN_ManuCycle  := FALSE,
              xIN_Quit       := xIN_Quit,
              xIN_AlarmAktiv := HMI.xAlarm,
              xIN_DryCycle   := FALSE,
              enIN_State     := enIN_State,
              tIN_Timeout    := T#10S,
              xIN_On         := TRUE);

SIMU.iCompletionHMI[5]           := PRG.st125_aut.iCompletionPC;
PRG.st125_aut.iProcessTimeMili_1 := PERS.iStationTimeDef1[5];
PRG.st125_aut.iProcessTimeMili_2 := PERS.iStationTimeDef2[5];
PRG.st125_aut(xIN_Init       := HMI.enState = enState.StateINIT,
              xIN_Start      := HMI.btArMain[9].press,
              xIN_Step       := HMI.btArMain[1].rtrig,
              xIN_ManuCycle  := FALSE,
              xIN_ManuCycle  := FALSE,
              xIN_Quit       := xIN_Quit,
              xIN_AlarmAktiv := HMI.xAlarm,
              xIN_DryCycle   := FALSE,
              enIN_State     := enIN_State,
              tIN_Timeout    := T#10S,
              xIN_On         := TRUE);

SIMU.iCompletionHMI[6]           := PRG.st130_aut.iCompletionPC;
PRG.st130_aut.iProcessTimeMili_1 := PERS.iStationTimeDef1[6];
PRG.st130_aut.iProcessTimeMili_2 := PERS.iStationTimeDef2[6];
PRG.st130_aut(xIN_Init       := HMI.enState = enState.StateINIT,
              xIN_Start      := HMI.btArMain[9].press,
              xIN_Step       := HMI.btArMain[1].rtrig,
              xIN_ManuCycle  := FALSE,
              xIN_ManuCycle  := FALSE,
              xIN_Quit       := xIN_Quit,
              xIN_AlarmAktiv := HMI.xAlarm,
              xIN_DryCycle   := FALSE,
              enIN_State     := enIN_State,
              tIN_Timeout    := T#10S,
              xIN_On         := TRUE);

SIMU.iCompletionHMI[7]           := PRG.st135_aut.iCompletionPC;
PRG.st135_aut.iProcessTimeMili_1 := PERS.iStationTimeDef1[7];
PRG.st135_aut.iProcessTimeMili_2 := PERS.iStationTimeDef2[7];
PRG.st135_aut(xIN_Init       := HMI.enState = enState.StateINIT,
              xIN_Start      := HMI.btArMain[9].press,
              xIN_Step       := HMI.btArMain[1].rtrig,
              xIN_ManuCycle  := FALSE,
              xIN_ManuCycle  := FALSE,
              xIN_Quit       := xIN_Quit,
              xIN_AlarmAktiv := HMI.xAlarm,
              xIN_DryCycle   := FALSE,
              enIN_State     := enIN_State,
              tIN_Timeout    := T#10S,
              xIN_On         := TRUE);

SIMU.iCompletionHMI[8]           := PRG.st140_aut.iCompletionPC;
PRG.st140_aut.iProcessTimeMili_1 := PERS.iStationTimeDef1[8];
PRG.st140_aut.iProcessTimeMili_2 := PERS.iStationTimeDef2[8];
PRG.st140_aut(xIN_Init       := HMI.enState = enState.StateINIT,
              xIN_Start      := HMI.btArMain[9].press,
              xIN_Step       := HMI.btArMain[1].rtrig,
              xIN_ManuCycle  := FALSE,
              xIN_ManuCycle  := FALSE,
              xIN_Quit       := xIN_Quit,
              xIN_AlarmAktiv := HMI.xAlarm,
              xIN_DryCycle   := FALSE,
              enIN_State     := enIN_State,
              tIN_Timeout    := T#10S,
              xIN_On         := TRUE);

SIMU.iCompletionHMI[9]           := PRG.st145_aut.iCompletionPC;
PRG.st145_aut.iProcessTimeMili_1 := PERS.iStationTimeDef1[9];
PRG.st145_aut.iProcessTimeMili_2 := PERS.iStationTimeDef2[9];
PRG.st145_aut(xIN_Init       := HMI.enState = enState.StateINIT,
              xIN_Start      := HMI.btArMain[9].press,
              xIN_Step       := HMI.btArMain[1].rtrig,
              xIN_ManuCycle  := FALSE,
              xIN_ManuCycle  := FALSE,
              xIN_Quit       := xIN_Quit,
              xIN_AlarmAktiv := HMI.xAlarm,
              xIN_DryCycle   := FALSE,
              enIN_State     := enIN_State,
              tIN_Timeout    := T#10S,
              xIN_On         := TRUE);

SIMU.iCompletionHMI[10]          := PRG.st150_aut.iCompletionPC;
PRG.st150_aut.iProcessTimeMili_1 := PERS.iStationTimeDef1[10];
PRG.st150_aut.iProcessTimeMili_2 := PERS.iStationTimeDef2[10];
PRG.st150_aut(xIN_Init       := HMI.enState = enState.StateINIT,
              xIN_Start      := HMI.btArMain[9].press,
              xIN_Step       := HMI.btArMain[1].rtrig,
              xIN_ManuCycle  := FALSE,
              xIN_ManuCycle  := FALSE,
              xIN_Quit       := xIN_Quit,
              xIN_AlarmAktiv := HMI.xAlarm,
              xIN_DryCycle   := FALSE,
              enIN_State     := enIN_State,
              tIN_Timeout    := T#10S,
              xIN_On         := TRUE);

SIMU.iCompletionHMI[11]          := PRG.st155_aut.iCompletionPC;
PRG.st155_aut.iProcessTimeMili_1 := PERS.iStationTimeDef1[11];
PRG.st155_aut.iProcessTimeMili_2 := PERS.iStationTimeDef2[11];
PRG.st155_aut(xIN_Init       := HMI.enState = enState.StateINIT,
              xIN_Start      := HMI.btArMain[9].press,
              xIN_Step       := HMI.btArMain[1].rtrig,
              xIN_ManuCycle  := FALSE,
              xIN_ManuCycle  := FALSE,
              xIN_Quit       := xIN_Quit,
              xIN_AlarmAktiv := HMI.xAlarm,
              xIN_DryCycle   := FALSE,
              enIN_State     := enIN_State,
              tIN_Timeout    := T#10S,
              xIN_On         := TRUE);

SIMU.iCompletionHMI[12]          := PRG.st160_aut.iCompletionPC;
PRG.st160_aut.iProcessTimeMili_1 := PERS.iStationTimeDef1[12];
PRG.st160_aut.iProcessTimeMili_2 := PERS.iStationTimeDef2[12];
PRG.st160_aut(xIN_Init       := HMI.enState = enState.StateINIT,
              xIN_Start      := HMI.btArMain[9].press,
              xIN_Step       := HMI.btArMain[1].rtrig,
              xIN_ManuCycle  := FALSE,
              xIN_ManuCycle  := FALSE,
              xIN_Quit       := xIN_Quit,
              xIN_AlarmAktiv := HMI.xAlarm,
              xIN_DryCycle   := FALSE,
              enIN_State     := enIN_State,
              tIN_Timeout    := T#10S,
              xIN_On         := TRUE);

SIMU.iCompletionHMI[13]          := PRG.st165_aut.iCompletionPC;
PRG.st165_aut.iProcessTimeMili_1 := PERS.iStationTimeDef1[13];
PRG.st165_aut.iProcessTimeMili_2 := PERS.iStationTimeDef2[13];
PRG.st165_aut(xIN_Init       := HMI.enState = enState.StateINIT,
              xIN_Start      := HMI.btArMain[9].press,
              xIN_Step       := HMI.btArMain[1].rtrig,
              xIN_ManuCycle  := FALSE,
              xIN_ManuCycle  := FALSE,
              xIN_Quit       := xIN_Quit,
              xIN_AlarmAktiv := HMI.xAlarm,
              xIN_DryCycle   := FALSE,
              enIN_State     := enIN_State,
              tIN_Timeout    := T#10S,
              xIN_On         := TRUE);

SIMU.iCompletionHMI[14]          := PRG.st170_aut.iCompletionPC;
PRG.st170_aut.iProcessTimeMili_1 := PERS.iStationTimeDef1[14];
PRG.st170_aut.iProcessTimeMili_2 := PERS.iStationTimeDef2[14];
PRG.st170_aut(xIN_Init       := HMI.enState = enState.StateINIT,
              xIN_Start      := HMI.btArMain[9].press,
              xIN_Step       := HMI.btArMain[1].rtrig,
              xIN_ManuCycle  := FALSE,
              xIN_ManuCycle  := FALSE,
              xIN_Quit       := xIN_Quit,
              xIN_AlarmAktiv := HMI.xAlarm,
              xIN_DryCycle   := FALSE,
              enIN_State     := enIN_State,
              tIN_Timeout    := T#10S,
              xIN_On         := TRUE);

SIMU.iCompletionHMI[15]          := PRG.st175_aut.iCompletionPC;
PRG.st175_aut.iProcessTimeMili_1 := PERS.iStationTimeDef1[15];
PRG.st175_aut.iProcessTimeMili_2 := PERS.iStationTimeDef2[15];
PRG.st175_aut(xIN_Init       := HMI.enState = enState.StateINIT,
              xIN_Start      := HMI.btArMain[9].press,
              xIN_Step       := HMI.btArMain[1].rtrig,
              xIN_ManuCycle  := FALSE,
              xIN_ManuCycle  := FALSE,
              xIN_Quit       := xIN_Quit,
              xIN_AlarmAktiv := HMI.xAlarm,
              xIN_DryCycle   := FALSE,
              enIN_State     := enIN_State,
              tIN_Timeout    := T#10S,
              xIN_On         := TRUE);

SIMU.iCompletionHMI[16]          := PRG.st176_aut.iCompletionPC;
PRG.st176_aut.iProcessTimeMili_1 := PERS.iStationTimeDef1[16];
PRG.st176_aut.iProcessTimeMili_2 := PERS.iStationTimeDef2[16];
PRG.st176_aut(xIN_Init       := HMI.enState = enState.StateINIT,
              xIN_Start      := HMI.btArMain[9].press,
              xIN_Step       := HMI.btArMain[1].rtrig,
              xIN_ManuCycle  := FALSE,
              xIN_ManuCycle  := FALSE,
              xIN_Quit       := xIN_Quit,
              xIN_AlarmAktiv := HMI.xAlarm,
              xIN_DryCycle   := FALSE,
              enIN_State     := enIN_State,
              tIN_Timeout    := T#10S,
              xIN_On         := TRUE);

SIMU.iCompletionHMI[17]          := PRG.st180_aut.iCompletionPC;
PRG.st180_aut.iProcessTimeMili_1 := PERS.iStationTimeDef1[17];
PRG.st180_aut.iProcessTimeMili_2 := PERS.iStationTimeDef2[17];
PRG.st180_aut(xIN_Init       := HMI.enState = enState.StateINIT,
              xIN_Start      := HMI.btArMain[9].press,
              xIN_Step       := HMI.btArMain[1].rtrig,
              xIN_ManuCycle  := FALSE,
              xIN_ManuCycle  := FALSE,
              xIN_Quit       := xIN_Quit,
              xIN_AlarmAktiv := HMI.xAlarm,
              xIN_DryCycle   := FALSE,
              enIN_State     := enIN_State,
              tIN_Timeout    := T#10S,
              xIN_On         := TRUE);

SIMU.iCompletionHMI[18]          := PRG.st185_aut.iCompletionPC;
PRG.st185_aut.iProcessTimeMili_1 := PERS.iStationTimeDef1[18];
PRG.st185_aut.iProcessTimeMili_2 := PERS.iStationTimeDef2[18];
PRG.st185_aut(xIN_Init       := HMI.enState = enState.StateINIT,
              xIN_Start      := HMI.btArMain[9].press,
              xIN_Step       := HMI.btArMain[1].rtrig,
              xIN_ManuCycle  := FALSE,
              xIN_ManuCycle  := FALSE,
              xIN_Quit       := xIN_Quit,
              xIN_AlarmAktiv := HMI.xAlarm,
              xIN_DryCycle   := FALSE,
              enIN_State     := enIN_State,
              tIN_Timeout    := T#10S,
              xIN_On         := TRUE);

END_PROGRAM

// ---- POUs/20_AUTO/ST100/FB_AUT_LOAD.TcPOU
FUNCTION_BLOCK FB_AUT_LOAD EXTENDS FB_AUT_ABSTRACT
    (****************************************************************************)
    (*	POU_AUT_zxx			Bausteinaufrufe Station	zxx							*)
    (*	Status				ungetestet											*)
    (*  Version:			1.0													*)
    (*	Beschrieb:																*)
    (*																			*)
    (*	Abläufe:			FB_ABLzxxA		Hauptablauf							*)
    (*																			*)
    (*																			*)
    (* 	25.09.2019/Dj															*)
    (****************************************************************************)
    (*	dd.mm.yyyy   KZ    x.y			Beschrieb								*)
    (****************************************************************************)
VAR_INPUT
    (* spezifische Eingänge *)

END_VAR
VAR_OUTPUT
    (* spezifische Ausgänge *)

END_VAR
VAR
    (* Bausteine *)
    _FB_ABL_100A : FB_ABL_LOAD;
END_VAR

(*******************************************************************)
(* Timer *)
(*******************************************************************)

(*******************************************************************)
(* Flanken / Merker *)
(*******************************************************************)
//MANU CYCLE
IF (enIN_State = StateMANU) AND xIN_ManuCycle THEN
    xManuCycle := TRUE;
END_IF;

IF (enIN_State <> StateMANU) OR xOUT_Done THEN
    xManuCycle := FALSE;
END_IF

//NEXT STEP
xNextStep := (enIN_State > StateSTEP) OR
             ((enIN_State = StateSTEP) AND xIN_Step) OR
             ((enIN_State = StateMANU) AND xManuCycle);

//RESET
xReset := ((enIN_State < StateREADY) AND (enIN_State <> StateINIT)) OR
          ((enIN_State = StateMANU) AND NOT xManuCycle);

(*******************************************************************)
(* Bausteinaufrufe Abläufe *)
(*******************************************************************)

_FB_ABL_100A(xIN_Reset    := xReset,
             xIN_Init     := xIN_Init,
             xIN_Quit     := xIN_Quit,
             xIN_Start    := enIN_State = enState.StateAUTO, //AND _FB_ABL_100A.xOUT_Done AND _FB_ABL_100A.xOUT_Ready,
             xIN_Sperre   := NOT xIN_On,
             xIN_NextStep := xNextStep,
             xIN_AlarmAktiv
                 := xIN_AlarmAktiv,
             xIN_DryCycle    := xIN_DryCycle,
             xIN_RestartCYCL := enIN_State = enState.StateAUTO, // only restart when the mover has move out
             enIN_State      := enIN_State,
             tIN_Timeout     := tIN_Timeout,
             pxFG_Freigabe   := ADR(xDummy),
             Mover           := THIS^.Mover,
             xOUT_ErrFlag    =>,
             xOUT_Busy       =>,
             xOUT_Done       =>,
             xOUT_Timeout    =>,
             xOUT_InitDone   =>,
             xOUT_Wait       =>,
             iOUT_Step       =>,
             bOUT_Error      =>);

(*******************************************************************)
(* Mover reset flags *)
(*******************************************************************)

(*******************************************************************)
(* OUTPUT *)
(*******************************************************************)
xOUT_InitDone := _FB_ABL_100A.xOUT_InitDone;
xOUT_Ready    := xOUT_InitDone;
xOUT_Done     := _FB_ABL_100A.xOUT_Done;
xOUT_ErrFlag  := _FB_ABL_100A.xOUT_ErrFlag;
xOUT_Wait     := _FB_ABL_100A.xOUT_Wait;
xOUT_AlarmST  := xOUT_ErrFlag;

(*******************************************************************)
(* Bausteinaufruf Error Station *)
(*******************************************************************)
// POU_ERR_VORLAGE(xIN_QUIT:=xIN_Quit , pstrArIN_ALARM:=ADR(HMI.strArALARM[1]));

METHOD GiveMover : IProcessSampleMover
VAR_INPUT
	mover : REFERENCE TO FB_Mover;
END_VAR
IF __ISVALIDREF(mover) THEN
    THIS^.Mover                       REF= mover;
END_IF
END_METHOD

(* % of completion of the process *)
PROPERTY iCompletionPC : INT
GET
iCompletionPC := THIS^._FB_ABL_100A.iOUT_ProcessCompletion;
END_GET
END_PROPERTY

(* Process time, expressed in milisecond *)
PROPERTY iProcessTimeMili_1 : DINT
GET
iProcessTimeMili_1 := TO_DINT(this^._FB_ABL_100A.iProcessTimeMili1);
END_GET
SET
THIS^._FB_ABL_100A.iProcessTimeMili1 := TO_UDINT(iProcessTimeMili_1);
END_SET
END_PROPERTY

(* Process time, expressed in milisecond *)
PROPERTY iProcessTimeMili_2 : DINT
GET
iProcessTimeMili_2 := TO_DINT(this^._FB_ABL_100A.iProcessTimeMili2);
END_GET
SET
THIS^._FB_ABL_100A.iProcessTimeMili2 := TO_UDINT(iProcessTimeMili_2);
END_SET
END_PROPERTY

PROPERTY ProcessExecution : ProcessExecution_e
GET
ProcessExecution := THIS^._ProcessExecution;
END_GET
SET
THIS^._ProcessExecution := ProcessExecution;
END_SET
END_PROPERTY

METHOD TakeMover : IProcessSampleMover
VAR_INPUT
END_VAR
THIS^.Mover REF= 0;
END_METHOD

PROPERTY xBusy : BOOL
GET
xBusy := This^._FB_ABL_100A.xOUT_Busy;
END_GET
SET
END_SET
END_PROPERTY

PROPERTY xDone : BOOL
GET
xDone := THIS^._FB_ABL_100A.xOUT_Ready OR THIS^._FB_ABL_100A.xOUT_Done;
END_GET
END_PROPERTY

PROPERTY xMoverPathFree : BOOL
GET
xMoverPathFree := THIS^._FB_ABL_100A.xOUT_MoverFree OR THIS^._FB_ABL_100A.xOUT_Ready OR THIS^._FB_ABL_100A.xOUT_Done;
END_GET
END_PROPERTY

PROPERTY xMoverShouldLeave : BOOL
GET
xMoverShouldLeave := THIS^._FB_ABL_100A.iOUT_Step = ST100_Load_e.SYNC_MOVER_LEAVE;
END_GET
END_PROPERTY

END_FUNCTION_BLOCK

// ---- POUs/20_AUTO/ST100/FB_ABL_LOAD.TcPOU
FUNCTION_BLOCK FB_ABL_LOAD
(****************************************************************************************)
(*	TITEL				Bezeichnung Ablauf	    										*)
(*	Status				ungetestet                         								*)
(*  Version:			1.0																*)
(*	Beschrieb:			Ablaufbeschreibung												*)
(*																						*)
(*	Steps:																				*)
(*		RESET:=0		Reset der Station												*)
(* 		INIT:=100		Initialisieren													*)
(*		... 			...																*)
(*		READY:=999		Initialisiert, Bereit für Start									*)
(*		START:=1000		Start Zyklisch 													*)
(*		... 			...																*)
(*		DONE:=8000		Letzer Schritt													*)
(*		ERROR:=9000		ALARM/Fehler													*)
(* 	09.09.2019/Dj																		*)
(***********************************Revisionen*******************************************)
(*	dd.mm.yyyy   KZ    x.y			Beschrieb											*)
(****************************************************************************************)

VAR_INPUT
    xIN_Reset       : BOOL;          // Schrittkette zurücksetzen 
    xIN_Init        : BOOL;          // Initialisieren
    xIN_Quit        : BOOL;          // Fehler quittieren 
    xIN_Start       : BOOL;          // Startbefehl
    xIN_Sperre      : BOOL;          // FB Sperren 
    xIN_NextStep    : BOOL;          // Nächsten Schritt ausführen 
    xIN_AlarmAktiv  : BOOL;          // Anlage hat Alarm
    xIN_DryCycle    : BOOL;          // Fahren ohne Teile
    xIN_RestartCYCL : BOOL;          // Zyklus erneut starten im STEP, END, LEERFAHREN
    enIN_State      : enState;       // Status Anlage
    tIN_Timeout     : TIME := T#10s; // Timout

    pxFG_Freigabe : POINTER TO BOOL; //Freigabe von Station

    // Application specific
    iProcessTimeMili1 : UDINT := 5000; // user defined station duration, in milisecond
    iProcessTimeMili2 : UDINT := 5000; // user defined station duration, in milisecond
    Mover            : REFERENCE TO FB_Mover;
    //xIN_MoverInPos  : BOOL;          // Set this flag when a mover is in position and ready to be handled
END_VAR
VAR_OUTPUT
    (* standart Ausgänge *)
    xOUT_ErrFlag     : BOOL;   // Error Flag 
    xOUT_Busy        : BOOL;   // Baustein befindet sich im Ablauf 
    xOUT_Done        : BOOL;   // Baustein hat den Ablauf beendet 		
    xOUT_Ready       : BOOL;   // Ready to begin, should be the same state as done	
    xOUT_Timeout     : BOOL;   // Timeout FB 
    xOUT_InitDone    : BOOL;   // initialisierung fertig
    xOUT_Wait        : BOOL;   // Wartet auf Bedingung
    iOUT_Step        : INT;    // Aktueller Schritt 
    sOUT_Step        : STRING; // Aktueller Schritt but in string format
    bOUT_Error       : BYTE;   // Fehlernummer

    iOUT_ProcessCompletion : INT; //process completion, express in % (0-100)
    xOUT_MoverFree   : BOOL;   // The mover is free to move
    //xOUT_MoverNeeded : BOOL;   // A mover is needed by this station to continue its process
END_VAR
VAR
    (* Standard *)
    (* Schritt *)
    iLastStep : INT; // Merker letzter Schritt 
    iPreStep  : INT; // Schritt zurück nach Alarm 
    iAktStep  : INT; // aktueller Schritt

    // Trigger Starten 
    rtSTART : R_TRIG;
    // Timer TimeOut 
    TON_Timeout : TON;

    (* Bausteine *)

    (* Spezial *)
    iStartProcessTimeMili : UDINT; // start of the processing time, accurate at 100ns 

END_VAR
VAR CONSTANT
END_VAR

(*******************************************************************)
(* Trigger  *)
(*******************************************************************)
(* Zurücksetzen *)
IF xIN_RESET THEN
    iPreStep  := ST100_Load_e.RESET;
    iOUT_Step := ST100_Load_e.RESET;
END_IF;

(* Error Quittieren *)
IF (bOUT_Error <> 0) AND xIN_Quit THEN
    xOUT_ErrFlag := FALSE;
    bOUT_Error   := 0;
    iOUT_Step    := iPreStep;
END_IF;

(*******************************************************************)
(* Timer *)
(*******************************************************************)
TON_Timeout(IN := xIN_NextStep AND (iLastStep = iOUT_Step) (*todo FG *) ,
            PT := tIN_Timeout);

(*******************************************************************)
(* Bausteine *)
(*******************************************************************)

(*******************************************************************)
(* OUTPUTS *)
(*******************************************************************)
// Error Flag 
xOUT_ErrFlag := (bOUT_Error <> 0);
// Baustein befindet sich im Ablauf 
xOUT_Busy := (iOUT_Step > ST100_Load_e.READY) AND (iOUT_Step < ST100_Load_e.DONE);
// Baustein hat den Ablauf beendet
xOUT_Done := (iOUT_Step = ST100_Load_e.DONE);
// Process ready
xOUT_Ready := (iOUT_Step = ST100_Load_e.READY);
// Timeout FB 				 		
xOUT_Timeout := TON_Timeout.Q;
// Itialisierung fertig			
xOUT_InitDone := (iOUT_Step = ST100_Load_e.READY);
// Aktueller Schritt			
iOUT_Step := iOUT_Step; //Im Ablauf gesetzt		
sOUT_Step := TO_STRING(iOUT_Step);
//Fehlernummer	 
bOUT_Error := bOUT_Error; //Im Ablauf/FB gesetzt	
(* Warte (alle Schritte wo auf FG oder Teile gewartet wird) *)
xOUT_Wait := (iOUT_Step = ST100_Load_e.DONE);

xOUT_MoverFree := iOUT_Step >= ST100_Load_e.MOVER_FREE_OP AND iOUT_Step < ST100_Load_e.MOVER_NEEDED_OP;

iOUT_ProcessCompletion := F_GetPercent(iAktStep,
                                       ST100_Load_e.START,
                                       ST100_Load_e.DONE,
                                       ST100_Load_e.proceedOperation_1,
                                       ST100_Load_e.proceedOperation_2,
                                       iStartProcessTimeMili,
                                       TO_DINT(iProcessTimeMili1),
                                       TO_DINT(iProcessTimeMili2));

(*******************************************************************)
(* Ablauf *)
(*******************************************************************)

(* Sperren *)
IF xIN_Sperre THEN
    iPreStep  := ST100_Load_e.RESET;
    iOUT_Step := ST100_Load_e.RESET;
    RETURN;
END_IF;

(* Schritt Merker *)
IF iAktStep <> iOUT_Step THEN
    iLastStep := iAktStep;
    iAktStep  := iOUT_Step;
END_IF

(* START *)
rtSTART(CLK := xIN_Start);

(*******************************************************************)
(* Schrittkette  *)
(*******************************************************************)
CASE iOUT_Step OF

(***** RESET *****)
ST100_Load_e.RESET: (* Schritt 0-99 *)
    //Initialisierungen
    //Start Init Ablauf
    IF xIN_Init THEN
        iOUT_Step := ST100_Load_e.INIT;
        //Start Manu Ablauf
    ELSIF enIN_State = StateMANU AND xIN_NextStep THEN
        iOUT_Step := ST100_Load_e.INIT;
    END_IF;

(***** INIT *****)
ST100_Load_e.INIT: (* Grundstellung ? *)
    IF TRUE THEN
        iOUT_Step := ST100_Load_e.READY;
    ELSE
        iOUT_Step := ST100_Load_e.INIT;
    END_IF;

(***** READY / INIT DONE *****)
ST100_Load_e.READY:   (* Start AUTO,END,LEER,STEP *)
    IF xIN_Start THEN //IF rtSTART.Q THEN
        iOUT_Step := ST100_Load_e.START;
    END_IF

(***** START  ZYKLISCH *****)
ST100_Load_e.START: (*  *)
    IF xIN_NextStep AND pxFG_Freigabe^ THEN
        iOUT_Step             := ST100_Load_e.proceedOperation_1;
        iStartProcessTimeMili := GetTick();
    END_IF;

ST100_Load_e.proceedOperation_1: (*  *)
    IF xIN_NextStep AND (GetTick() - iStartProcessTimeMili) >= (iProcessTimeMili1) THEN
        iOUT_Step := ST100_Load_e.waitOnMover;
    END_IF;

ST100_Load_e.waitOnMover: (*  *)
    IF xIN_NextStep AND __ISVALIDREF(Mover) THEN
        iStartProcessTimeMili := GetTick();
        iOUT_Step             := ST100_Load_e.proceedOperation_2;
    END_IF;

ST100_Load_e.proceedOperation_2: (*  *)
    IF xIN_NextStep AND (GetTick() - iStartProcessTimeMili) >= (iProcessTimeMili2) THEN
        iOUT_Step := ST100_Load_e.SYNC_MOVER_LEAVE;
    END_IF;

ST100_Modify_e.SYNC_MOVER_LEAVE:
    // The mover needs to be taken by MoverMan
    IF NOT __ISVALIDREF(Mover) THEN
        iOUT_Step := ST100_Unload_e.DONE;
    END_IF

(***** DONE *****)
ST100_Load_e.DONE: (* Letzter Schritt  *)
    IF NOT xIN_AlarmAktiv THEN
        //AUTO
        IF (enIN_State = StateAUTO) AND xIN_RestartCYCL THEN
            iOUT_Step := ST100_Load_e.START;
            //STEP / END / LEERFAHREN restart
        ELSIF (enIN_State < StateAUTO) AND (enIN_State >= enState.StateSTEP) AND xIN_RestartCYCL THEN
            iOUT_Step := ST100_Load_e.START;
            //STEP / END / LEERFAHREN fertig
        ELSIF (enIN_State = StateREADY) THEN
            iOUT_Step := ST100_Load_e.READY;
        END_IF;
    END_IF;

(************ ERROR *************)
ST100_Load_e.ERROR: (* ERROR *) ;

END_CASE;

END_FUNCTION_BLOCK

// ---- POUs/20_AUTO/ST100/F_GetPercent.TcPOU
FUNCTION F_GetPercent : INT
VAR_INPUT
    iAktStep   : INT; // actual step
    iStepStart : INT; // step start
    iStepDone  : INT; // step stop
    iStepP1    : INT; // step process 1
    iStepP2    : INT; // step process 2

    uiStartProcessTimeMili : UDINT;
    diProcessTimeDuration1 : DINT;
    diProcessTimeDuration2 : DINT;
END_VAR
VAR
END_VAR


IF iAktStep < iStepStart THEN
    F_GetPercent := 0;
ELSIF iStepDone = iAktStep THEN
    F_GetPercent := 100;
ELSE
    // F_GetPercent := getPercent(iAktStep, TO_INT(iStepStart), TO_INT(caca.releaseMover) + 1);
    IF diProcessTimeDuration1 > 0 AND diProcessTimeDuration2 > 0 THEN
        IF iAktStep < iStepP1 THEN
            F_GetPercent := 0;
        ELSIF iAktStep > iStepP2 THEN
            F_GetPercent := 100;
        ELSIF iAktStep = iStepP1 THEN
            F_GetPercent := TO_INT((TO_DINT(GetTick() - uiStartProcessTimeMili) * 50) / diProcessTimeDuration1);
        ELSIF iAktStep = iStepP2 THEN
            F_GetPercent :=
                50 + TO_INT((TO_DINT(GetTick() - uiStartProcessTimeMili) * 50) / diProcessTimeDuration2);
        ELSE
            F_GetPercent := 50;
        END_IF
    ELSE
        F_GetPercent := 0;
    END_IF
END_IF

END_FUNCTION

// ---- POUs/20_AUTO/ST100/FB_AUT_UNLOAD.TcPOU
FUNCTION_BLOCK FB_AUT_UNLOAD EXTENDS FB_AUT_ABSTRACT
(****************************************************************************)
(*	POU_AUT_zxx			Bausteinaufrufe Station	zxx							*)
(*	Status				ungetestet											*)
(*  Version:			1.0													*)
(*	Beschrieb:																*)
(*																			*)
(*	Abläufe:			FB_ABLzxxA		Hauptablauf							*)
(*																			*)
(*																			*)
(* 	25.09.2019/Dj															*)
(****************************************************************************)
(*	dd.mm.yyyy   KZ    x.y			Beschrieb								*)
(****************************************************************************)
VAR_INPUT
    (* spezifische Eingänge *)

END_VAR
VAR_OUTPUT
    (* spezifische Ausgänge *)

END_VAR
VAR
    (* Bausteine *)
    _FB_ABL_100A : FB_ABL_UNLOAD;
END_VAR

(*******************************************************************)
(* Timer *)
(*******************************************************************)

(*******************************************************************)
(* Flanken / Merker *)
(*******************************************************************)
//MANU CYCLE
IF (enIN_State = StateMANU) AND xIN_ManuCycle THEN
    xManuCycle := TRUE;
END_IF;

IF (enIN_State <> StateMANU) OR xOUT_Done THEN
    xManuCycle := FALSE;
END_IF

//NEXT STEP
xNextStep := (enIN_State > StateSTEP) OR
             ((enIN_State = StateSTEP) AND xIN_Step) OR
             ((enIN_State = StateMANU) AND xManuCycle);

//RESET
xReset := ((enIN_State < StateREADY) AND (enIN_State <> StateINIT)) OR
          ((enIN_State = StateMANU) AND NOT xManuCycle);

(*******************************************************************)
(* Bausteinaufrufe Abläufe *)
(*******************************************************************)

_FB_ABL_100A(xIN_Reset    := xReset,
             xIN_Init     := xIN_Init,
             xIN_Quit     := xIN_Quit,
             xIN_Start    := enIN_State = enState.StateAUTO, //AND _FB_ABL_100A.xOUT_Done AND _FB_ABL_100A.xOUT_Ready,
             xIN_Sperre   := NOT xIN_On,
             xIN_NextStep := xNextStep,
             xIN_AlarmAktiv
                 := xIN_AlarmAktiv,
             xIN_DryCycle    := xIN_DryCycle,
             xIN_RestartCYCL := enIN_State = enState.StateAUTO, // only restart when the mover has move out
             enIN_State      := enIN_State,
             tIN_Timeout     := tIN_Timeout,
             pxFG_Freigabe   := ADR(xDummy),
             Mover           := THIS^.Mover,
             xOUT_ErrFlag    =>,
             xOUT_Busy       =>,
             xOUT_Done       =>,
             xOUT_Timeout    =>,
             xOUT_InitDone   =>,
             xOUT_Wait       =>,
             iOUT_Step       =>,
             bOUT_Error      =>);

(*******************************************************************)
(* Mover reset flags *)
(*******************************************************************)

(*******************************************************************)
(* OUTPUT *)
(*******************************************************************)
xOUT_InitDone := _FB_ABL_100A.xOUT_InitDone;
xOUT_Ready    := xOUT_InitDone;
xOUT_Done     := _FB_ABL_100A.xOUT_Done;
xOUT_ErrFlag  := _FB_ABL_100A.xOUT_ErrFlag;
xOUT_Wait     := _FB_ABL_100A.xOUT_Wait;
xOUT_AlarmST  := xOUT_ErrFlag;

(*******************************************************************)
(* Bausteinaufruf Error Station *)
(*******************************************************************)
// POU_ERR_VORLAGE(xIN_QUIT:=xIN_Quit , pstrArIN_ALARM:=ADR(HMI.strArALARM[1]));

METHOD GiveMover : IProcessSampleMover
VAR_INPUT
	mover : REFERENCE TO FB_Mover;
END_VAR
IF __ISVALIDREF(mover) THEN
    THIS^.Mover REF= mover;
END_IF
END_METHOD

(* % of completion of the process *)
PROPERTY iCompletionPC : INT
GET
iCompletionPC := THIS^._FB_ABL_100A.iOUT_ProcessCompletion;
END_GET
END_PROPERTY

(* Process time, expressed in milisecond *)
PROPERTY iProcessTimeMili_1 : DINT
GET
iProcessTimeMili_1 := TO_DINT(this^._FB_ABL_100A.iProcessTimeMili1);
END_GET
SET
THIS^._FB_ABL_100A.iProcessTimeMili1 := TO_UDINT(iProcessTimeMili_1);
END_SET
END_PROPERTY

(* Process time, expressed in milisecond *)
PROPERTY iProcessTimeMili_2 : DINT
GET
iProcessTimeMili_2 := TO_DINT(this^._FB_ABL_100A.iProcessTimeMili2);
END_GET
SET
THIS^._FB_ABL_100A.iProcessTimeMili2 := TO_UDINT(iProcessTimeMili_2);
END_SET
END_PROPERTY

PROPERTY ProcessExecution : ProcessExecution_e
GET
ProcessExecution := THIS^._ProcessExecution;
END_GET
SET
THIS^._ProcessExecution := ProcessExecution;
END_SET
END_PROPERTY

METHOD TakeMover : IProcessSampleMover
VAR_INPUT
END_VAR
THIS^.Mover REF= 0;
END_METHOD

PROPERTY xBusy : BOOL
GET
xBusy := This^._FB_ABL_100A.xOUT_Busy;
END_GET
SET
END_SET
END_PROPERTY

PROPERTY xDone : BOOL
GET
xDone := THIS^._FB_ABL_100A.xOUT_Ready OR THIS^._FB_ABL_100A.xOUT_Done;
END_GET
END_PROPERTY

PROPERTY xMoverPathFree : BOOL
GET
xMoverPathFree := THIS^._FB_ABL_100A.xOUT_MoverFree OR THIS^._FB_ABL_100A.xOUT_Ready OR THIS^._FB_ABL_100A.xOUT_Done;
END_GET
END_PROPERTY

PROPERTY xMoverShouldLeave : BOOL
GET
xMoverShouldLeave := THIS^._FB_ABL_100A.iOUT_Step = ST100_Unload_e.SYNC_MOVER_LEAVE;
END_GET
END_PROPERTY

END_FUNCTION_BLOCK

// ---- POUs/20_AUTO/ST100/FB_ABL_UNLOAD.TcPOU
FUNCTION_BLOCK FB_ABL_UNLOAD
(****************************************************************************************)
(*	TITEL				Bezeichnung Ablauf	    										*)
(*	Status				ungetestet                         								*)
(*  Version:			1.0																*)
(*	Beschrieb:			Ablaufbeschreibung												*)
(*																						*)
(*	Steps:																				*)
(*		RESET:=0		Reset der Station												*)
(* 		INIT:=100		Initialisieren													*)
(*		... 			...																*)
(*		READY:=999		Initialisiert, Bereit für Start									*)
(*		START:=1000		Start Zyklisch 													*)
(*		... 			...																*)
(*		DONE:=8000		Letzer Schritt													*)
(*		ERROR:=9000		ALARM/Fehler													*)
(* 	09.09.2019/Dj																		*)
(***********************************Revisionen*******************************************)
(*	dd.mm.yyyy   KZ    x.y			Beschrieb											*)
(****************************************************************************************)

VAR_INPUT
    xIN_Reset       : BOOL;          // Schrittkette zurücksetzen 
    xIN_Init        : BOOL;          // Initialisieren
    xIN_Quit        : BOOL;          // Fehler quittieren 
    xIN_Start       : BOOL;          // Startbefehl
    xIN_Sperre      : BOOL;          // FB Sperren 
    xIN_NextStep    : BOOL;          // Nächsten Schritt ausführen 
    xIN_AlarmAktiv  : BOOL;          // Anlage hat Alarm
    xIN_DryCycle    : BOOL;          // Fahren ohne Teile
    xIN_RestartCYCL : BOOL;          // Zyklus erneut starten im STEP, END, LEERFAHREN
    enIN_State      : enState;       // Status Anlage
    tIN_Timeout     : TIME := T#10s; // Timout

    pxFG_Freigabe : POINTER TO BOOL; //Freigabe von Station

    // Application specific
    iProcessTimeMili1 : UDINT := 5000; // user defined station duration, in milisecond
    iProcessTimeMili2 : UDINT := 5000; // user defined station duration, in milisecond
    Mover            : REFERENCE TO FB_Mover;
    //xIN_MoverInPos  : BOOL;          // Set this flag when a mover is in position and ready to be handled
END_VAR
VAR_OUTPUT
    (* standart Ausgänge *)
    xOUT_ErrFlag     : BOOL;   // Error Flag 
    xOUT_Busy        : BOOL;   // Baustein befindet sich im Ablauf 
    xOUT_Done        : BOOL;   // Baustein hat den Ablauf beendet 		
    xOUT_Ready       : BOOL;   // Ready to begin, should be the same state as done	
    xOUT_Timeout     : BOOL;   // Timeout FB 
    xOUT_InitDone    : BOOL;   // initialisierung fertig
    xOUT_Wait        : BOOL;   // Wartet auf Bedingung
    xOUT_MoverFree   : BOOL;   // The mover is free to move
    //xOUT_MoverNeeded : BOOL;   // A mover is needed by this station to continue its process
    iOUT_Step        : INT;    // Aktueller Schritt 
    sOUT_Step        : STRING; // Aktueller Schritt but in string format
    bOUT_Error       : BYTE;   // Fehlernummer

    iOUT_ProcessCompletion : INT; //process completion, express in % (0-100)
END_VAR
VAR
    (* Standard *)
    (* Schritt *)
    iLastStep : INT; // Merker letzter Schritt 
    iPreStep  : INT; // Schritt zurück nach Alarm 
    iAktStep  : INT; // aktueller Schritt

    // Trigger Starten 
    rtSTART : R_TRIG;
    // Timer TimeOut 
    TON_Timeout : TON;

    (* Bausteine *)

    (* Spezial *)
    iStartProcessTimeMili : UDINT; // start of the processing time, accurate at 100ns 

END_VAR
VAR CONSTANT
END_VAR

(*******************************************************************)
(* Trigger  *)
(*******************************************************************)
(* Zurücksetzen *)
IF xIN_RESET THEN
    iPreStep  := ST100_Unload_e.RESET;
    iOUT_Step := ST100_Unload_e.RESET;
END_IF;

(* Error Quittieren *)
IF (bOUT_Error <> 0) AND xIN_Quit THEN
    xOUT_ErrFlag := FALSE;
    bOUT_Error   := 0;
    iOUT_Step    := iPreStep;
END_IF;

(*******************************************************************)
(* Timer *)
(*******************************************************************)
TON_Timeout(IN := xIN_NextStep AND (iLastStep = iOUT_Step) (*todo FG *) ,
            PT := tIN_Timeout);

(*******************************************************************)
(* Bausteine *)
(*******************************************************************)

(*******************************************************************)
(* OUTPUTS *)
(*******************************************************************)
// Error Flag 
xOUT_ErrFlag := (bOUT_Error <> 0);
// Baustein befindet sich im Ablauf 
xOUT_Busy := (iOUT_Step > ST100_Unload_e.READY) AND (iOUT_Step < ST100_Unload_e.DONE);
// Baustein hat den Ablauf beendet
xOUT_Done := (iOUT_Step = ST100_Unload_e.DONE);
// Process ready
xOUT_Ready := (iOUT_Step = ST100_Unload_e.READY);
// Timeout FB 				 		
xOUT_Timeout := TON_Timeout.Q;
// Itialisierung fertig			
xOUT_InitDone := (iOUT_Step = ST100_Unload_e.READY);
// Aktueller Schritt			
iOUT_Step := iOUT_Step; //Im Ablauf gesetzt		
sOUT_Step := TO_STRING(iOUT_Step);
//Fehlernummer	 
bOUT_Error := bOUT_Error; //Im Ablauf/FB gesetzt	
(* Warte (alle Schritte wo auf FG oder Teile gewartet wird) *)
xOUT_Wait := (iOUT_Step = ST100_Unload_e.DONE);

xOUT_MoverFree := NOT (iOUT_Step >= ST100_Unload_e.MOVER_NEEDED_OP AND iOUT_Step < ST100_Unload_e.MOVER_FREE_OP);

iOUT_ProcessCompletion := F_GetPercent(iAktStep,
                                       ST100_Unload_e.START,
                                       ST100_Unload_e.DONE,
                                       ST100_Unload_e.proceedOperation_1,
                                       ST100_Unload_e.proceedOperation_2,
                                       iStartProcessTimeMili,
                                       TO_DINT(iProcessTimeMili1),
                                       TO_DINT(iProcessTimeMili2));

(*******************************************************************)
(* Ablauf *)
(*******************************************************************)

(* Sperren *)
IF xIN_Sperre THEN
    iPreStep  := ST100_Unload_e.RESET;
    iOUT_Step := ST100_Unload_e.RESET;
    RETURN;
END_IF;

(* Schritt Merker *)
IF iAktStep <> iOUT_Step THEN
    iLastStep := iAktStep;
    iAktStep  := iOUT_Step;
END_IF

(* START *)
rtSTART(CLK := xIN_Start);

(*******************************************************************)
(* Schrittkette  *)
(*******************************************************************)
CASE iOUT_Step OF

(***** RESET *****)
ST100_Unload_e.RESET: (* Schritt 0-99 *)
    //Initialisierungen
    //Start Init Ablauf
    IF xIN_Init THEN
        iOUT_Step := ST100_Unload_e.INIT;
        //Start Manu Ablauf
    ELSIF enIN_State = StateMANU AND xIN_NextStep THEN
        iOUT_Step := ST100_Unload_e.INIT;
    END_IF;

(***** INIT *****)
ST100_Unload_e.INIT: (* Grundstellung ? *)
    IF TRUE THEN
        iOUT_Step := ST100_Unload_e.READY;
    ELSE
        iOUT_Step := ST100_Unload_e.INIT;
    END_IF;

(***** READY / INIT DONE *****)
ST100_Unload_e.READY: (* Start AUTO,END,LEER,STEP *)
    IF xIN_Start THEN //IF rtSTART.Q THEN
        iOUT_Step := ST100_Unload_e.START;
    END_IF

(***** START  ZYKLISCH *****)
ST100_Unload_e.START: (*  *)
    IF xIN_NextStep AND pxFG_Freigabe^ THEN
        iOUT_Step := ST100_Unload_e.waitOnMover;
    END_IF;

ST100_Unload_e.waitOnMover: (*  *)
    IF xIN_NextStep AND __ISVALIDREF(Mover) THEN
        iStartProcessTimeMili := GetTick();
        iOUT_Step             := ST100_Unload_e.proceedOperation_1;
    END_IF;

ST100_Unload_e.proceedOperation_1: (*  *)
    IF xIN_NextStep AND (GetTick() - iStartProcessTimeMili) >= (iProcessTimeMili1) THEN
        iOUT_Step := ST100_Unload_e.SYNC_MOVER_LEAVE;
    END_IF;

ST100_Unload_e.SYNC_MOVER_LEAVE:
    // The mover needs to be taken by MoverMan
    IF NOT __ISVALIDREF(Mover) THEN
        iStartProcessTimeMili := GetTick();
        iOUT_Step             := ST100_Unload_e.proceedOperation_2;
    END_IF

ST100_Unload_e.proceedOperation_2: (*  *)
    IF xIN_NextStep AND (GetTick() - iStartProcessTimeMili) >= (iProcessTimeMili2) THEN
        iOUT_Step := ST100_Unload_e.DONE;
    END_IF;

(***** DONE *****)
ST100_Unload_e.DONE: (* Letzter Schritt  *)
    IF NOT xIN_AlarmAktiv THEN
        //AUTO
        IF (enIN_State = StateAUTO) AND xIN_RestartCYCL THEN
            iOUT_Step := ST100_Unload_e.START;
            //STEP / END / LEERFAHREN restart
        ELSIF (enIN_State < StateAUTO) AND (enIN_State >= enState.StateSTEP) AND xIN_RestartCYCL THEN
            iOUT_Step := ST100_Unload_e.START;
            //STEP / END / LEERFAHREN fertig
        ELSIF (enIN_State = StateREADY) THEN
            iOUT_Step := ST100_Unload_e.READY;
        END_IF;
    END_IF;

(************ ERROR *************)
ST100_Unload_e.ERROR: (* ERROR *) ;

END_CASE;

END_FUNCTION_BLOCK

// ---- POUs/20_AUTO/ST100/FB_AUT_MODIFY.TcPOU
FUNCTION_BLOCK FB_AUT_MODIFY EXTENDS FB_AUT_ABSTRACT
    (****************************************************************************)
    (*	POU_AUT_zxx			Bausteinaufrufe Station	zxx							*)
    (*	Status				ungetestet											*)
    (*  Version:			1.0													*)
    (*	Beschrieb:																*)
    (*																			*)
    (*	Abläufe:			FB_ABLzxxA		Hauptablauf							*)
    (*																			*)
    (*																			*)
    (* 	25.09.2019/Dj															*)
    (****************************************************************************)
    (*	dd.mm.yyyy   KZ    x.y			Beschrieb								*)
    (****************************************************************************)
VAR_INPUT
    (* spezifische Eingänge *)

END_VAR
VAR_OUTPUT
    (* spezifische Ausgänge *)

END_VAR
VAR
    (* Bausteine *)
    _FB_ABL_100A : FB_ABL_MODIFY;
END_VAR

(*******************************************************************)
(* Timer *)
(*******************************************************************)

(*******************************************************************)
(* Flanken / Merker *)
(*******************************************************************)
//MANU CYCLE
IF (enIN_State = StateMANU) AND xIN_ManuCycle THEN
    xManuCycle := TRUE;
END_IF;

IF (enIN_State <> StateMANU) OR xOUT_Done THEN
    xManuCycle := FALSE;
END_IF

//NEXT STEP
xNextStep := (enIN_State > StateSTEP) OR
             ((enIN_State = StateSTEP) AND xIN_Step) OR
             ((enIN_State = StateMANU) AND xManuCycle);

//RESET
xReset := ((enIN_State < StateREADY) AND (enIN_State <> StateINIT)) OR
          ((enIN_State = StateMANU) AND NOT xManuCycle);

(*******************************************************************)
(* Bausteinaufrufe Abläufe *)
(*******************************************************************)

_FB_ABL_100A(xIN_Reset    := xReset,
             xIN_Init     := xIN_Init,
             xIN_Quit     := xIN_Quit,
             xIN_Start    := enIN_State = enState.StateAUTO, //AND _FB_ABL_100A.xOUT_Done AND _FB_ABL_100A.xOUT_Ready,
             xIN_Sperre   := NOT xIN_On,
             xIN_NextStep := xNextStep,
             xIN_AlarmAktiv
                 := xIN_AlarmAktiv,
             xIN_DryCycle    := xIN_DryCycle,
             xIN_RestartCYCL := enIN_State = enState.StateAUTO, // only restart when the mover has move out
             enIN_State      := enIN_State,
             tIN_Timeout     := tIN_Timeout,
             pxFG_Freigabe   := ADR(xDummy),
             Mover           := THIS^.Mover,
             xOUT_ErrFlag    =>,
             xOUT_Busy       =>,
             xOUT_Done       =>,
             xOUT_Timeout    =>,
             xOUT_InitDone   =>,
             xOUT_Wait       =>,
             iOUT_Step       =>,
             bOUT_Error      =>);

(*******************************************************************)
(* Mover reset flags *)
(*******************************************************************)

(*******************************************************************)
(* OUTPUT *)
(*******************************************************************)
xOUT_InitDone := _FB_ABL_100A.xOUT_InitDone;
xOUT_Ready    := xOUT_InitDone;
xOUT_Done     := _FB_ABL_100A.xOUT_Done;
xOUT_ErrFlag  := _FB_ABL_100A.xOUT_ErrFlag;
xOUT_Wait     := _FB_ABL_100A.xOUT_Wait;
xOUT_AlarmST  := xOUT_ErrFlag;

(*******************************************************************)
(* Bausteinaufruf Error Station *)
(*******************************************************************)
// POU_ERR_VORLAGE(xIN_QUIT:=xIN_Quit , pstrArIN_ALARM:=ADR(HMI.strArALARM[1]));

METHOD GiveMover : IProcessSampleMover
VAR_INPUT
	mover : REFERENCE TO FB_Mover;
END_VAR
IF __ISVALIDREF(mover) THEN
    THIS^.Mover                       REF= mover;
END_IF
END_METHOD

(* % of completion of the process *)
PROPERTY iCompletionPC : INT
GET
iCompletionPC := THIS^._FB_ABL_100A.iOUT_ProcessCompletion;
END_GET
END_PROPERTY

(* Process time, expressed in milisecond *)
PROPERTY iProcessTimeMili_1 : DINT
GET
iProcessTimeMili_1 := TO_DINT(this^._FB_ABL_100A.iProcessTimeMili1);
END_GET
SET
THIS^._FB_ABL_100A.iProcessTimeMili1 := TO_UDINT(iProcessTimeMili_1);
END_SET
END_PROPERTY

(* Process time, expressed in milisecond *)
PROPERTY iProcessTimeMili_2 : DINT
GET
iProcessTimeMili_2 := TO_DINT(this^._FB_ABL_100A.iProcessTimeMili2);
END_GET
SET
THIS^._FB_ABL_100A.iProcessTimeMili2 := TO_UDINT(iProcessTimeMili_2);
END_SET
END_PROPERTY

PROPERTY ProcessExecution : ProcessExecution_e
GET
ProcessExecution := THIS^._ProcessExecution;
END_GET
SET
THIS^._ProcessExecution := ProcessExecution;
END_SET
END_PROPERTY

METHOD TakeMover : IProcessSampleMover
VAR_INPUT
END_VAR
THIS^.Mover REF= 0;
END_METHOD

PROPERTY xBusy : BOOL
GET
xBusy := This^._FB_ABL_100A.xOUT_Busy;
END_GET
SET
END_SET
END_PROPERTY

PROPERTY xDone : BOOL
GET
xDone := THIS^._FB_ABL_100A.xOUT_Ready OR THIS^._FB_ABL_100A.xOUT_Done;
END_GET
END_PROPERTY

PROPERTY xMoverPathFree : BOOL
GET
xMoverPathFree := THIS^._FB_ABL_100A.xOUT_MoverFree OR THIS^._FB_ABL_100A.xOUT_Ready OR THIS^._FB_ABL_100A.xOUT_Done;
END_GET
END_PROPERTY

PROPERTY xMoverShouldLeave : BOOL
GET
xMoverShouldLeave := THIS^._FB_ABL_100A.iOUT_Step = ST100_Modify_e.SYNC_MOVER_LEAVE;
END_GET
END_PROPERTY

END_FUNCTION_BLOCK

// ---- POUs/20_AUTO/ST100/FB_ABL_MODIFY.TcPOU
FUNCTION_BLOCK FB_ABL_MODIFY
(****************************************************************************************)
(*	TITEL				Bezeichnung Ablauf	    										*)
(*	Status				ungetestet                         								*)
(*  Version:			1.0																*)
(*	Beschrieb:			Ablaufbeschreibung												*)
(*																						*)
(*	Steps:																				*)
(*		RESET:=0		Reset der Station												*)
(* 		INIT:=100		Initialisieren													*)
(*		... 			...																*)
(*		READY:=999		Initialisiert, Bereit für Start									*)
(*		START:=1000		Start Zyklisch 													*)
(*		... 			...																*)
(*		DONE:=8000		Letzer Schritt													*)
(*		ERROR:=9000		ALARM/Fehler													*)
(* 	09.09.2019/Dj																		*)
(***********************************Revisionen*******************************************)
(*	dd.mm.yyyy   KZ    x.y			Beschrieb											*)
(****************************************************************************************)

VAR_INPUT
    xIN_Reset       : BOOL;          // Schrittkette zurücksetzen 
    xIN_Init        : BOOL;          // Initialisieren
    xIN_Quit        : BOOL;          // Fehler quittieren 
    xIN_Start       : BOOL;          // Startbefehl
    xIN_Sperre      : BOOL;          // FB Sperren 
    xIN_NextStep    : BOOL;          // Nächsten Schritt ausführen 
    xIN_AlarmAktiv  : BOOL;          // Anlage hat Alarm
    xIN_DryCycle    : BOOL;          // Fahren ohne Teile
    xIN_RestartCYCL : BOOL;          // Zyklus erneut starten im STEP, END, LEERFAHREN
    enIN_State      : enState;       // Status Anlage
    tIN_Timeout     : TIME := T#10s; // Timout

    pxFG_Freigabe : POINTER TO BOOL; //Freigabe von Station

    // Application specific
    iProcessTimeMili1 : UDINT := 5000; // user defined station duration, in milisecond
    iProcessTimeMili2 : UDINT := 5000; // user defined station duration, in milisecond
    Mover            : REFERENCE TO FB_Mover;
    //xIN_MoverInPos  : BOOL;          // Set this flag when a mover is in position and ready to be handled
END_VAR
VAR_OUTPUT
    (* standart Ausgänge *)
    xOUT_ErrFlag     : BOOL;   // Error Flag 
    xOUT_Busy        : BOOL;   // Baustein befindet sich im Ablauf 
    xOUT_Done        : BOOL;   // Baustein hat den Ablauf beendet 		
    xOUT_Ready       : BOOL;   // Ready to begin, should be the same state as done	
    xOUT_Timeout     : BOOL;   // Timeout FB 
    xOUT_InitDone    : BOOL;   // initialisierung fertig
    xOUT_Wait        : BOOL;   // Wartet auf Bedingung
    iOUT_Step        : INT;    // Aktueller Schritt 
    sOUT_Step        : STRING; // Aktueller Schritt but in string format
    bOUT_Error       : BYTE;   // Fehlernummer

    xOUT_MoverFree   : BOOL;   // The mover is free to move
    //xOUT_MoverNeeded : BOOL;   // A mover is needed by this station to continue its process
    iOUT_ProcessCompletion : INT; //process completion, express in % (0-100)
END_VAR
VAR
    (* Standard *)
    (* Schritt *)
    iLastStep : INT; // Merker letzter Schritt 
    iPreStep  : INT; // Schritt zurück nach Alarm 
    iAktStep  : INT; // aktueller Schritt

    // Trigger Starten 
    rtSTART : R_TRIG;
    // Timer TimeOut 
    TON_Timeout : TON;

    (* Bausteine *)

    (* Spezial *)
    iStartProcessTimeMili : UDINT; // start of the processing time, accurate at 100ns 
	
	_bBewegung : BOOL;
	_bBewegungDist : INT := 20;

END_VAR
VAR CONSTANT
END_VAR

(*******************************************************************)
(* Trigger  *)
(*******************************************************************)
(* Zurücksetzen *)
IF xIN_RESET THEN
    iPreStep  := ST100_Modify_e.RESET;
    iOUT_Step := ST100_Modify_e.RESET;
END_IF;

(* Error Quittieren *)
IF (bOUT_Error <> 0) AND xIN_Quit THEN
    xOUT_ErrFlag := FALSE;
    bOUT_Error   := 0;
    iOUT_Step    := iPreStep;
END_IF;

(*******************************************************************)
(* Timer *)
(*******************************************************************)
TON_Timeout(IN := xIN_NextStep AND (iLastStep = iOUT_Step) (*todo FG *) ,
            PT := tIN_Timeout);

(*******************************************************************)
(* Bausteine *)
(*******************************************************************)

(*******************************************************************)
(* OUTPUTS *)
(*******************************************************************)
// Error Flag 
xOUT_ErrFlag := (bOUT_Error <> 0);
// Baustein befindet sich im Ablauf 
xOUT_Busy := (iOUT_Step > ST100_Modify_e.READY) AND (iOUT_Step < ST100_Modify_e.DONE);
// Baustein hat den Ablauf beendet
xOUT_Done := (iOUT_Step = ST100_Modify_e.DONE);
// Process ready
xOUT_Ready := (iOUT_Step = ST100_Modify_e.READY);
// Timeout FB 				 		
xOUT_Timeout := TON_Timeout.Q;
// Itialisierung fertig			
xOUT_InitDone := (iOUT_Step = ST100_Modify_e.READY);
// Aktueller Schritt			
iOUT_Step := iOUT_Step; //Im Ablauf gesetzt		
sOUT_Step := TO_STRING(iOUT_Step);
//Fehlernummer	 
bOUT_Error := bOUT_Error; //Im Ablauf/FB gesetzt	
(* Warte (alle Schritte wo auf FG oder Teile gewartet wird) *)
xOUT_Wait := (iOUT_Step = ST100_Modify_e.DONE);

xOUT_MoverFree := iOUT_Step = ST100_Modify_e.waitOnMover;

iOUT_ProcessCompletion := F_GetPercent(iAktStep,
                                       ST100_Modify_e.START,
                                       ST100_Modify_e.DONE,
                                       ST100_Modify_e.proceedOperation_1,
                                       ST100_Modify_e.proceedOperation_2,
                                       iStartProcessTimeMili,
                                       TO_DINT(iProcessTimeMili1),
                                       TO_DINT(iProcessTimeMili2));

(*******************************************************************)
(* Ablauf *)
(*******************************************************************)

(* Sperren *)
IF xIN_Sperre THEN
    iPreStep  := ST100_Modify_e.RESET;
    iOUT_Step := ST100_Modify_e.RESET;
    RETURN;
END_IF;

(* Schritt Merker *)
IF iAktStep <> iOUT_Step THEN
    iLastStep := iAktStep;
    iAktStep  := iOUT_Step;
END_IF

(* START *)
rtSTART(CLK := xIN_Start);

(*******************************************************************)
(* Schrittkette  *)
(*******************************************************************)
CASE iOUT_Step OF

(***** RESET *****)
ST100_Modify_e.RESET: (* Schritt 0-99 *)
    //Initialisierungen
    //Start Init Ablauf
    IF xIN_Init THEN
        iOUT_Step := ST100_Modify_e.INIT;
        //Start Manu Ablauf
    ELSIF enIN_State = StateMANU AND xIN_NextStep THEN
        iOUT_Step := ST100_Modify_e.INIT;
    END_IF;

(***** INIT *****)
ST100_Modify_e.INIT: (* Grundstellung ? *)
    IF TRUE THEN
        iOUT_Step := ST100_Modify_e.READY;
    ELSE
        iOUT_Step := ST100_Modify_e.INIT;
    END_IF;

(***** READY / INIT DONE *****)
ST100_Modify_e.READY: (* Start AUTO,END,LEER,STEP *)
    IF xIN_Start THEN //IF rtSTART.Q THEN
        iOUT_Step := ST100_Modify_e.START;
    END_IF

(***** START  ZYKLISCH *****)
ST100_Modify_e.START: (*  *)
    IF xIN_NextStep AND pxFG_Freigabe^ THEN
        iOUT_Step             := ST100_Modify_e.waitOnMover;
        iStartProcessTimeMili := GetTick();
    END_IF;

ST100_Modify_e.waitOnMover: (*  *)
    IF xIN_NextStep AND __ISVALIDREF(Mover) THEN
        iStartProcessTimeMili := GetTick();
        iOUT_Step             := ST100_Modify_e.proceedOperation_1;
    END_IF;

ST100_Modify_e.proceedOperation_1: (*  *)
    IF xIN_NextStep AND (GetTick() - iStartProcessTimeMili) >= (iProcessTimeMili1) THEN
        iStartProcessTimeMili := GetTick();
        iOUT_Step             := ST100_Modify_e.proceedOperation_2;
		_bBewegung := FALSE;
		
    ELSIF __ISVALIDREF(Mover) THEN
        IF Mover.MoverAxis.isInPos THEN
            IF _bBewegung THEN
               // Mover.MoverAxis.RelMoveTo(_bBewegungDist);
            ELSE
                //Mover.MoverAxis.RelMoveTo(-_bBewegungDist);
            END_IF

            _bBewegung := NOT _bBewegung;
        END_IF;
    END_IF;

ST100_Modify_e.proceedOperation_2: (*  *)
    IF xIN_NextStep AND (GetTick() - iStartProcessTimeMili) >= (iProcessTimeMili2) THEN
        iOUT_Step := ST100_Modify_e.SYNC_MOVER_LEAVE;
    END_IF;

ST100_Modify_e.SYNC_MOVER_LEAVE:
    // The mover needs to be taken by MoverMan
    IF NOT __ISVALIDREF(Mover) THEN
        iOUT_Step := ST100_Unload_e.DONE;
    END_IF

(***** DONE *****)
ST100_Modify_e.DONE: (* Letzter Schritt  *)
    IF NOT xIN_AlarmAktiv THEN
        //AUTO
        IF (enIN_State = StateAUTO) AND xIN_RestartCYCL THEN
            iOUT_Step := ST100_Modify_e.START;
            //STEP / END / LEERFAHREN restart
        ELSIF (enIN_State < StateAUTO) AND (enIN_State >= enState.StateSTEP) AND xIN_RestartCYCL THEN
            iOUT_Step := ST100_Modify_e.START;
            //STEP / END / LEERFAHREN fertig
        ELSIF (enIN_State = StateREADY) THEN
            iOUT_Step := ST100_Modify_e.READY;
        END_IF;
    END_IF;

(************ ERROR *************)
ST100_Modify_e.ERROR: (* ERROR *) ;

END_CASE;

END_FUNCTION_BLOCK

// ---- POUs/20_AUTO/FileMan/FB_FileMan.TcPOU
FUNCTION_BLOCK FB_FileMan
VAR_INPUT
    sPathName   : STRING; //
    bSave       : BOOL;
    bLoad       : BOOL;
    sRefString  : POINTER TO STRING(2000);
    uiStringLen : DINT; // string length
END_VAR
VAR_OUTPUT
    bError   : BOOL;  // true when a FB is in error (all fb are mixed here)
    nErrorId : UDINT; // the error id from the fb in error (all fb are mixed here)

    currentState : INT; // current state of this FB, use it for debug
END_VAR
VAR
    fb_open  : FB_FileOpen;
    fb_write : FB_FileWrite;
    fb_read  : FB_FileRead;
    fb_close : FB_FileClose;
    hFile    : UINT; // file number holder for write operation
    state    : INT := 0;

    bOpState : INT;   //0 = saving operation, 1 = loading operation, other = error
    nMode    : DWORD; // file open monde, depending on the command

    byteRead : UDINT; //number of byte read so far
END_VAR


CASE state OF

0: (* wait for operation *)
    IF bSave THEN
        state    := 1;
        bOpState := 0;
        nMode    := FOPEN_MODEWRITE;
    ELSIF bLoad THEN
        state    := 1;
        bOpState := 1;
        nMode    := FOPEN_MODEREAD;
    END_IF

1: (* open *)
    fb_open(sNetId    := '',
            sPathName := sPathName,
            nMode     := nMode,
            ePath     := PATH_GENERIC,
            bExecute  := TRUE,
            tTimeout  := T#3S,
            bBusy     =>,
            bError    =>,
            nErrId    =>,
            hFile     => hFile);

    IF NOT fb_open.bBusy THEN
        fb_open(bExecute := FALSE);

        IF 0 = bOpState THEN
            state := 3;
        ELSIF 1 = bOpState THEN
            state    := 5;
            byteRead := 0;
        END_IF
    END_IF

3: (* write *)
    fb_write(sNetId     := '',
             hFile      := hFile,
             pWriteBuff := sRefString,
             cbWriteLen := TO_UDINT(uiStringLen),
             bExecute   := TRUE,
             tTimeout   := T#3S,
             bBusy      =>,
             bError     =>,
             nErrId     =>,
             cbWrite    =>);

    IF NOT fb_write.bBusy THEN
        fb_write(bExecute := FALSE);
        state := 10;
    END_IF

